REGION Network 7: 380A1 FB
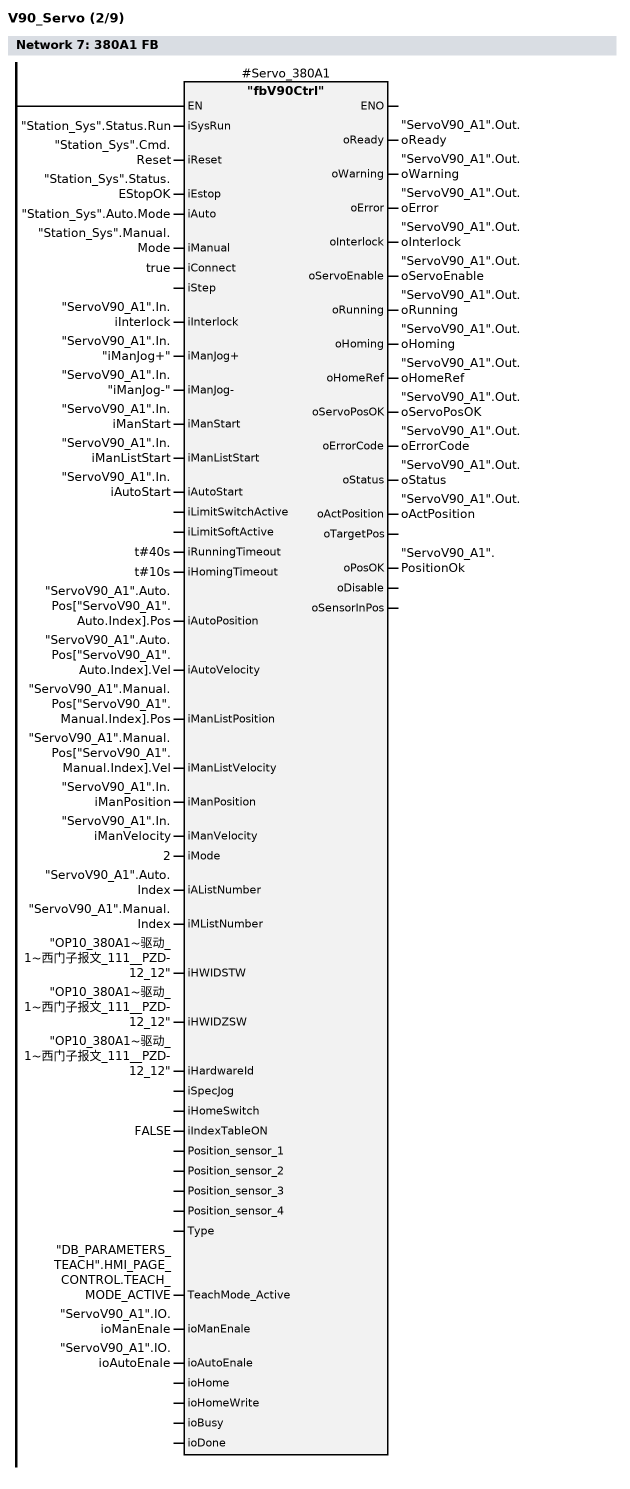
   RUNG wire#powerrail
      #Servo_380A1(iSysRun := "Station_Sys".Status.Run, iReset := "Station_Sys".Cmd.Reset, iEstop := "Station_Sys".Status.EStopOK, iAuto := "Station_Sys".Auto.Mode, iManual := "Station_Sys".Manual.Mode, iConnect := true, iStep :=, iInterlock := "ServoV90_A1".In.iInterlock, "iManJog+" := "ServoV90_A1".In."iManJog+", "iManJog-" := "ServoV90_A1".In."iManJog-", iManStart := "ServoV90_A1".In.iManStart, iManListStart := "ServoV90_A1".In.iManListStart, iAutoStart := "ServoV90_A1".In.iAutoStart, iLimitSwitchActive :=, iLimitSoftActive :=, iRunningTimeout := t#40s, iHomingTimeout := t#10s, iAutoPosition := "ServoV90_A1".Auto.Pos["ServoV90_A1".Auto.Index].Pos, iAutoVelocity := "ServoV90_A1".Auto.Pos["ServoV90_A1".Auto.Index].Vel, iManListPosition := "ServoV90_A1".Manual.Pos["ServoV90_A1".Manual.Index].Pos, iManListVelocity := "ServoV90_A1".Manual.Pos["ServoV90_A1".Manual.Index].Vel, iManPosition := "ServoV90_A1".In.iManPosition, iManVelocity := "ServoV90_A1".In.iManVelocity, iMode := 2, iAListNumber := "ServoV90_A1".Auto.Index, iMListNumber := "ServoV90_A1".Manual.Index, iHWIDSTW := "OP10_380A1~驱动_1~西门子报文_111__PZD-12_12", iHWIDZSW := "OP10_380A1~驱动_1~西门子报文_111__PZD-12_12", iHardwareId := "OP10_380A1~驱动_1~西门子报文_111__PZD-12_12", iSpecJog :=, iHomeSwitch :=, iIndexTableON := FALSE, Position_sensor_1 :=, Position_sensor_2 :=, Position_sensor_3 :=, Position_sensor_4 :=, "Type" :=, TeachMode_Active := "DB_PARAMETERS_TEACH".HMI_PAGE_CONTROL.TEACH_MODE_ACTIVE, ioManEnale := "ServoV90_A1".IO.ioManEnale, ioAutoEnale := "ServoV90_A1".IO.ioAutoEnale, ioHome :=, ioHomeWrite :=, ioBusy :=, ioDone :=, oReady => "ServoV90_A1".Out.oReady, oWarning => "ServoV90_A1".Out.oWarning, oError => "ServoV90_A1".Out.oError, oInterlock => "ServoV90_A1".Out.oInterlock, oServoEnable => "ServoV90_A1".Out.oServoEnable, oRunning => "ServoV90_A1".Out.oRunning, oHoming => "ServoV90_A1".Out.oHoming, oHomeRef => "ServoV90_A1".Out.oHomeRef, oServoPosOK => "ServoV90_A1".Out.oServoPosOK, oErrorCode => "ServoV90_A1".Out.oErrorCode, oStatus => "ServoV90_A1".Out.oStatus, oActPosition => "ServoV90_A1".Out.oActPosition, oTargetPos =>, oPosOK => "ServoV90_A1".PositionOk, oDisable =>, oSensorInPos =>)
   END_RUNG
   // the same network as SCL:
   #Servo_380A1(iSysRun := "Station_Sys".Status.Run,   // "fbV90Ctrl"
                iReset := "Station_Sys".Cmd.Reset,
                iEstop := "Station_Sys".Status.EStopOK,
                iAuto := "Station_Sys".Auto.Mode,
                iManual := "Station_Sys".Manual.Mode,
                iConnect := true,
                iInterlock := "ServoV90_A1".In.iInterlock,
                "iManJog+" := "ServoV90_A1".In."iManJog+",
                "iManJog-" := "ServoV90_A1".In."iManJog-",
                iManStart := "ServoV90_A1".In.iManStart,
                iManListStart := "ServoV90_A1".In.iManListStart,
                iAutoStart := "ServoV90_A1".In.iAutoStart,
                iRunningTimeout := t#40s,
                iHomingTimeout := t#10s,
                iAutoPosition := "ServoV90_A1".Auto.Pos["ServoV90_A1".Auto.Index].Pos,
                iAutoVelocity := "ServoV90_A1".Auto.Pos["ServoV90_A1".Auto.Index].Vel,
                iManListPosition := "ServoV90_A1".Manual.Pos["ServoV90_A1".Manual.Index].Pos,
                iManListVelocity := "ServoV90_A1".Manual.Pos["ServoV90_A1".Manual.Index].Vel,
                iManPosition := "ServoV90_A1".In.iManPosition,
                iManVelocity := "ServoV90_A1".In.iManVelocity,
                iMode := 2,
                iAListNumber := "ServoV90_A1".Auto.Index,
                iMListNumber := "ServoV90_A1".Manual.Index,
                iHWIDSTW := "OP10_380A1~驱动_1~西门子报文_111__PZD-12_12",
                iHWIDZSW := "OP10_380A1~驱动_1~西门子报文_111__PZD-12_12",
                iHardwareId := "OP10_380A1~驱动_1~西门子报文_111__PZD-12_12",
                iIndexTableON := FALSE,
                TeachMode_Active := "DB_PARAMETERS_TEACH".HMI_PAGE_CONTROL.TEACH_MODE_ACTIVE,
                ioManEnale := "ServoV90_A1".IO.ioManEnale,
                ioAutoEnale := "ServoV90_A1".IO.ioAutoEnale,
                oReady => "ServoV90_A1".Out.oReady,
                oWarning => "ServoV90_A1".Out.oWarning,
                oError => "ServoV90_A1".Out.oError,
                oInterlock => "ServoV90_A1".Out.oInterlock,
                oServoEnable => "ServoV90_A1".Out.oServoEnable,
                oRunning => "ServoV90_A1".Out.oRunning,
                oHoming => "ServoV90_A1".Out.oHoming,
                oHomeRef => "ServoV90_A1".Out.oHomeRef,
                oServoPosOK => "ServoV90_A1".Out.oServoPosOK,
                oErrorCode => "ServoV90_A1".Out.oErrorCode,
                oStatus => "ServoV90_A1".Out.oStatus,
                oActPosition => "ServoV90_A1".Out.oActPosition,
                oPosOK => "ServoV90_A1".PositionOk);
END_REGION

REGION Network 8 (SCL): 故障显示 / Fault indication
   //"ST70_DeviceError".Servo1.ServoDriverError := "ServoV90_A1".Out.oError;
END_REGION

REGION Network 9: <<<<<<<<<<<<<<<<<<<<<381A1 Servo>>>>>>>>>>>>>>>>>>>>>>>>>
END_REGION

REGION Network 10: negtive motion/action/...automaticly
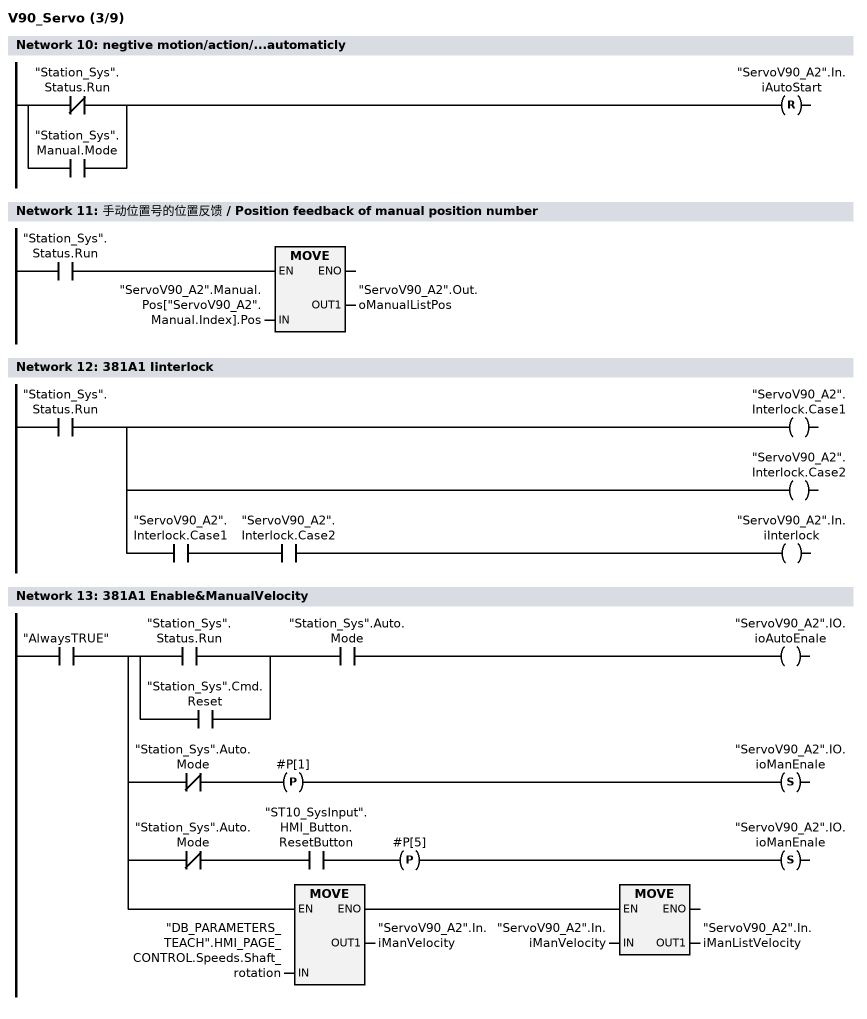
   RUNG wire#powerrail
      I_Contact( "Station_Sys".Status.Run )
      wire#w1
      R_Coil( "ServoV90_A2".In.iAutoStart )
   END_RUNG
   RUNG wire#powerrail
      Contact( "Station_Sys".Manual.Mode )
   END_RUNG wire#w1
   // the same network as SCL:
   IF NOT "Station_Sys".Status.Run OR "Station_Sys".Manual.Mode THEN
       "ServoV90_A2".In.iAutoStart := FALSE;
   END_IF;
END_REGION

REGION Network 11: 手动位置号的位置反馈 / Position feedback of manual position number
   RUNG wire#powerrail
      Contact( "Station_Sys".Status.Run )
      Move(in := "ServoV90_A2".Manual.Pos["ServoV90_A2".Manual.Index].Pos, out1 => "ServoV90_A2".Out.oManualListPos)
   END_RUNG
   // the same network as SCL:
   IF "Station_Sys".Status.Run THEN
       "ServoV90_A2".Out.oManualListPos := "ServoV90_A2".Manual.Pos["ServoV90_A2".Manual.Index].Pos;
   END_IF;
END_REGION

REGION Network 12: 381A1 Iinterlock
   RUNG wire#powerrail
      Contact( "Station_Sys".Status.Run )
      wire#w1
      Coil( "ServoV90_A2".Interlock.Case1 )
   END_RUNG
   RUNG wire#w1
      Coil( "ServoV90_A2".Interlock.Case2 )
   END_RUNG
   RUNG wire#w1
      Contact( "ServoV90_A2".Interlock.Case1 )
      Contact( "ServoV90_A2".Interlock.Case2 )
      Coil( "ServoV90_A2".In.iInterlock )
   END_RUNG
   // the same network as SCL:
   "ServoV90_A2".Interlock.Case1 := "Station_Sys".Status.Run;
   "ServoV90_A2".Interlock.Case2 := "Station_Sys".Status.Run;
   "ServoV90_A2".In.iInterlock := "Station_Sys".Status.Run AND "ServoV90_A2".Interlock.Case1 AND "ServoV90_A2".Interlock.Case2;
END_REGION

REGION Network 13: 381A1 Enable&ManualVelocity
   RUNG wire#powerrail
      Contact( "AlwaysTRUE" )
      wire#w1
      Contact( "Station_Sys".Status.Run )
      wire#w2
      Contact( "Station_Sys".Auto.Mode )
      Coil( "ServoV90_A2".IO.ioAutoEnale )
   END_RUNG
   RUNG wire#w1
      Contact( "Station_Sys".Cmd.Reset )
   END_RUNG wire#w2
   RUNG wire#w1
      I_Contact( "Station_Sys".Auto.Mode )
      P_Trig( #P[1] )
      S_Coil( "ServoV90_A2".IO.ioManEnale )
   END_RUNG
   RUNG wire#w1
      I_Contact( "Station_Sys".Auto.Mode )
      Contact( "ST10_SysInput".HMI_Button.ResetButton )
      P_Trig( #P[5] )
      S_Coil( "ServoV90_A2".IO.ioManEnale )
   END_RUNG
   RUNG wire#w1
      Move(in := "DB_PARAMETERS_TEACH".HMI_PAGE_CONTROL.Speeds.Shaft_rotation, out1 => "ServoV90_A2".In.iManVelocity)
      Move(in := "ServoV90_A2".In.iManVelocity, out1 => "ServoV90_A2".In.iManListVelocity)
   END_RUNG
   // the same network as SCL:
   "ServoV90_A2".IO.ioAutoEnale := "AlwaysTRUE" AND ("Station_Sys".Status.Run OR "Station_Sys".Cmd.Reset) AND "Station_Sys".Auto.Mode;
   #_w1 := "AlwaysTRUE" AND NOT "Station_Sys".Auto.Mode;
   #_w2 := #_w1 AND NOT #P[1];   // rising edge
   #P[1] := #_w1;
   IF #_w2 THEN "ServoV90_A2".IO.ioManEnale := TRUE; END_IF;
   #_w3 := "AlwaysTRUE" AND NOT "Station_Sys".Auto.Mode AND "ST10_SysInput".HMI_Button.ResetButton;
   #_w4 := #_w3 AND NOT #P[5];   // rising edge
   #P[5] := #_w3;
   IF #_w4 THEN "ServoV90_A2".IO.ioManEnale := TRUE; END_IF;
   IF "AlwaysTRUE" THEN
       "ServoV90_A2".In.iManVelocity := "DB_PARAMETERS_TEACH".HMI_PAGE_CONTROL.Speeds.Shaft_rotation;
       "ServoV90_A2".In.iManListVelocity := "ServoV90_A2".In.iManVelocity;
   END_IF;
END_REGION

REGION Network 14 (SCL): 381A1 RecipePosition
    IF "Station_Sys".Status.Run THEN
        "ServoV90_A2".Manual.Pos[1].Pos := "ServoV90_A2".Auto.Pos[1].Pos := REAL_TO_DINT("Parameter".AxisRun.Axis[2].Pos1.Position*1000);
       "ServoV90_A2".Manual.Pos[1].Vel := "ServoV90_A2".Auto.Pos[1].Vel := "Parameter".AxisRun.Axis[2].Pos1.Speed;

       "ServoV90_A2".Manual.Pos[2].Pos := "ServoV90_A2".Auto.Pos[2].Pos := REAL_TO_DINT("Parameter".AxisRun.Axis[2].Pos2.Position*1000);
       "ServoV90_A2".Manual.Pos[2].Vel := "ServoV90_A2".Auto.Pos[2].Vel := "Parameter".AxisRun.Axis[2].Pos2.Speed;

       "ServoV90_A2".Manual.Pos[3].Pos := "ServoV90_A2".Auto.Pos[3].Pos := REAL_TO_DINT("Parameter".AxisRun.Axis[2].Pos3.Position*1000);
       "ServoV90_A2".Manual.Pos[3].Vel := "ServoV90_A2".Auto.Pos[3].Vel := "Parameter".AxisRun.Axis[2].Pos3.Speed;

       "ServoV90_A2".Manual.Pos[4].Pos := "ServoV90_A2".Auto.Pos[4].Pos := REAL_TO_DINT("Parameter".AxisRun.Axis[2].Pos4.Position*1000);
       "ServoV90_A2".Manual.Pos[4].Vel := "ServoV90_A2".Auto.Pos[4].Vel := "Parameter".AxisRun.Axis[2].Pos4.Speed;

       "ServoV90_A2".Manual.Pos[5].Pos := "ServoV90_A2".Auto.Pos[5].Pos := REAL_TO_DINT("Parameter".AxisRun.Axis[2].Pos5.Position*1000);
       "ServoV90_A2".Manual.Pos[5].Vel := "ServoV90_A2".Auto.Pos[5].Vel := "Parameter".AxisRun.Axis[2].Pos5.Speed;

       "ServoV90_A2".Manual.Pos[6].Pos := "ServoV90_A2".Auto.Pos[6].Pos := REAL_TO_DINT("Parameter".AxisRun.Axis[2].Pos6.Position*1000);
       "ServoV90_A2".Manual.Pos[6].Vel := "ServoV90_A2".Auto.Pos[6].Vel := "Parameter".AxisRun.Axis[2].Pos6.Speed;

       "ServoV90_A2".Manual.Pos[7].Pos := "ServoV90_A2".Auto.Pos[7].Pos := REAL_TO_DINT("Parameter".AxisRun.Axis[2].Pos7.Position*1000);
       "ServoV90_A2".Manual.Pos[7].Vel := "ServoV90_A2".Auto.Pos[7].Vel := "Parameter".AxisRun.Axis[2].Pos7.Speed;

       "ServoV90_A2".Manual.Pos[8].Pos := "ServoV90_A2".Auto.Pos[8].Pos := REAL_TO_DINT("Parameter".AxisRun.Axis[2].Pos8.Position*1000);
       "ServoV90_A2".Manual.Pos[8].Vel := "ServoV90_A2".Auto.Pos[8].Vel := "Parameter".AxisRun.Axis[2].Pos8.Speed;

       "ServoV90_A2".Manual.Pos[9].Pos := "ServoV90_A2".Auto.Pos[9].Pos := REAL_TO_DINT("Parameter".AxisRun.Axis[2].Pos9.Position*1000);
       "ServoV90_A2".Manual.Pos[9].Vel := "ServoV90_A2".Auto.Pos[9].Vel := "Parameter".AxisRun.Axis[2].Pos9.Speed;

       "ServoV90_A2".Manual.Pos[10].Pos := "ServoV90_A2".Auto.Pos[10].Pos := REAL_TO_DINT("Parameter".AxisRun.Axis[2].Pos10.Position*1000);
       "ServoV90_A2".Manual.Pos[10].Vel := "ServoV90_A2".Auto.Pos[10].Vel := "Parameter".AxisRun.Axis[2].Pos10.Speed;
   END_IF;
END_REGION

REGION Network 15: 381A1 FB
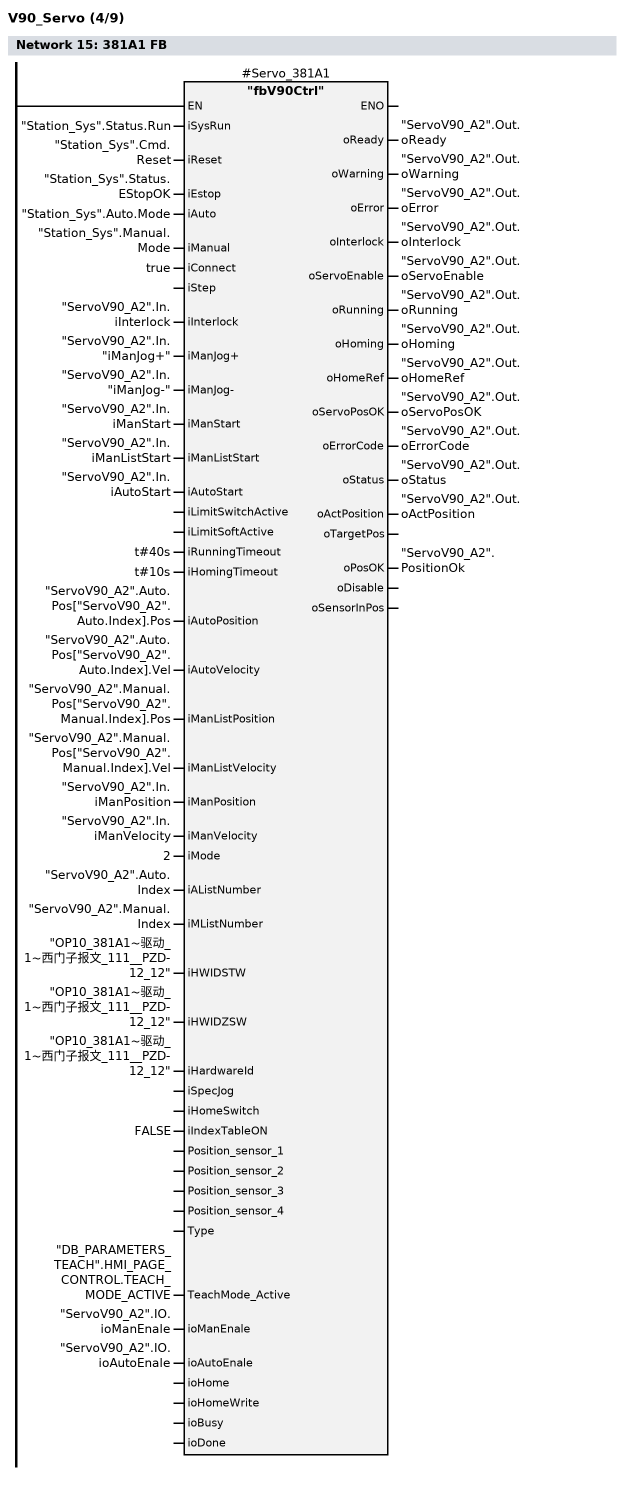
   RUNG wire#powerrail
      #Servo_381A1(iSysRun := "Station_Sys".Status.Run, iReset := "Station_Sys".Cmd.Reset, iEstop := "Station_Sys".Status.EStopOK, iAuto := "Station_Sys".Auto.Mode, iManual := "Station_Sys".Manual.Mode, iConnect := true, iStep :=, iInterlock := "ServoV90_A2".In.iInterlock, "iManJog+" := "ServoV90_A2".In."iManJog+", "iManJog-" := "ServoV90_A2".In."iManJog-", iManStart := "ServoV90_A2".In.iManStart, iManListStart := "ServoV90_A2".In.iManListStart, iAutoStart := "ServoV90_A2".In.iAutoStart, iLimitSwitchActive :=, iLimitSoftActive :=, iRunningTimeout := t#40s, iHomingTimeout := t#10s, iAutoPosition := "ServoV90_A2".Auto.Pos["ServoV90_A2".Auto.Index].Pos, iAutoVelocity := "ServoV90_A2".Auto.Pos["ServoV90_A2".Auto.Index].Vel, iManListPosition := "ServoV90_A2".Manual.Pos["ServoV90_A2".Manual.Index].Pos, iManListVelocity := "ServoV90_A2".Manual.Pos["ServoV90_A2".Manual.Index].Vel, iManPosition := "ServoV90_A2".In.iManPosition, iManVelocity := "ServoV90_A2".In.iManVelocity, iMode := 2, iAListNumber := "ServoV90_A2".Auto.Index, iMListNumber := "ServoV90_A2".Manual.Index, iHWIDSTW := "OP10_381A1~驱动_1~西门子报文_111__PZD-12_12", iHWIDZSW := "OP10_381A1~驱动_1~西门子报文_111__PZD-12_12", iHardwareId := "OP10_381A1~驱动_1~西门子报文_111__PZD-12_12", iSpecJog :=, iHomeSwitch :=, iIndexTableON := FALSE, Position_sensor_1 :=, Position_sensor_2 :=, Position_sensor_3 :=, Position_sensor_4 :=, "Type" :=, TeachMode_Active := "DB_PARAMETERS_TEACH".HMI_PAGE_CONTROL.TEACH_MODE_ACTIVE, ioManEnale := "ServoV90_A2".IO.ioManEnale, ioAutoEnale := "ServoV90_A2".IO.ioAutoEnale, ioHome :=, ioHomeWrite :=, ioBusy :=, ioDone :=, oReady => "ServoV90_A2".Out.oReady, oWarning => "ServoV90_A2".Out.oWarning, oError => "ServoV90_A2".Out.oError, oInterlock => "ServoV90_A2".Out.oInterlock, oServoEnable => "ServoV90_A2".Out.oServoEnable, oRunning => "ServoV90_A2".Out.oRunning, oHoming => "ServoV90_A2".Out.oHoming, oHomeRef => "ServoV90_A2".Out.oHomeRef, oServoPosOK => "ServoV90_A2".Out.oServoPosOK, oErrorCode => "ServoV90_A2".Out.oErrorCode, oStatus => "ServoV90_A2".Out.oStatus, oActPosition => "ServoV90_A2".Out.oActPosition, oTargetPos =>, oPosOK => "ServoV90_A2".PositionOk, oDisable =>, oSensorInPos =>)
   END_RUNG
   // the same network as SCL:
   #Servo_381A1(iSysRun := "Station_Sys".Status.Run,   // "fbV90Ctrl"
                iReset := "Station_Sys".Cmd.Reset,
                iEstop := "Station_Sys".Status.EStopOK,
                iAuto := "Station_Sys".Auto.Mode,
                iManual := "Station_Sys".Manual.Mode,
                iConnect := true,
                iInterlock := "ServoV90_A2".In.iInterlock,
                "iManJog+" := "ServoV90_A2".In."iManJog+",
                "iManJog-" := "ServoV90_A2".In."iManJog-",
                iManStart := "ServoV90_A2".In.iManStart,
                iManListStart := "ServoV90_A2".In.iManListStart,
                iAutoStart := "ServoV90_A2".In.iAutoStart,
                iRunningTimeout := t#40s,
                iHomingTimeout := t#10s,
                iAutoPosition := "ServoV90_A2".Auto.Pos["ServoV90_A2".Auto.Index].Pos,
                iAutoVelocity := "ServoV90_A2".Auto.Pos["ServoV90_A2".Auto.Index].Vel,
                iManListPosition := "ServoV90_A2".Manual.Pos["ServoV90_A2".Manual.Index].Pos,
                iManListVelocity := "ServoV90_A2".Manual.Pos["ServoV90_A2".Manual.Index].Vel,
                iManPosition := "ServoV90_A2".In.iManPosition,
                iManVelocity := "ServoV90_A2".In.iManVelocity,
                iMode := 2,
                iAListNumber := "ServoV90_A2".Auto.Index,
                iMListNumber := "ServoV90_A2".Manual.Index,
                iHWIDSTW := "OP10_381A1~驱动_1~西门子报文_111__PZD-12_12",
                iHWIDZSW := "OP10_381A1~驱动_1~西门子报文_111__PZD-12_12",
                iHardwareId := "OP10_381A1~驱动_1~西门子报文_111__PZD-12_12",
                iIndexTableON := FALSE,
                TeachMode_Active := "DB_PARAMETERS_TEACH".HMI_PAGE_CONTROL.TEACH_MODE_ACTIVE,
                ioManEnale := "ServoV90_A2".IO.ioManEnale,
                ioAutoEnale := "ServoV90_A2".IO.ioAutoEnale,
                oReady => "ServoV90_A2".Out.oReady,
                oWarning => "ServoV90_A2".Out.oWarning,
                oError => "ServoV90_A2".Out.oError,
                oInterlock => "ServoV90_A2".Out.oInterlock,
                oServoEnable => "ServoV90_A2".Out.oServoEnable,
                oRunning => "ServoV90_A2".Out.oRunning,
                oHoming => "ServoV90_A2".Out.oHoming,
                oHomeRef => "ServoV90_A2".Out.oHomeRef,
                oServoPosOK => "ServoV90_A2".Out.oServoPosOK,
                oErrorCode => "ServoV90_A2".Out.oErrorCode,
                oStatus => "ServoV90_A2".Out.oStatus,
                oActPosition => "ServoV90_A2".Out.oActPosition,
                oPosOK => "ServoV90_A2".PositionOk);
END_REGION

REGION Network 16 (SCL): 故障显示 / Fault indication
   //"ST70_DeviceError".Servo2.ServoDriverError := "ServoV90_A2".Out.oError;
   //

   "ServoV90_A3".Auto.Index := "ServoV90_A3".Auto.Index;
END_REGION

REGION Network 17: <<<<<<<<<<<<<<<<<<<<<382A1 Servo>>>>>>>>>>>>>>>>>>>>>>>>>
END_REGION

REGION Network 18: <<<<<<<<<<<<<<<<<<<<<382A1 Servo>>>>>>>>>>>>>>>>>>>>>>>>> / $$$$####### NEW TECHNOLOGY OBJECTS #################
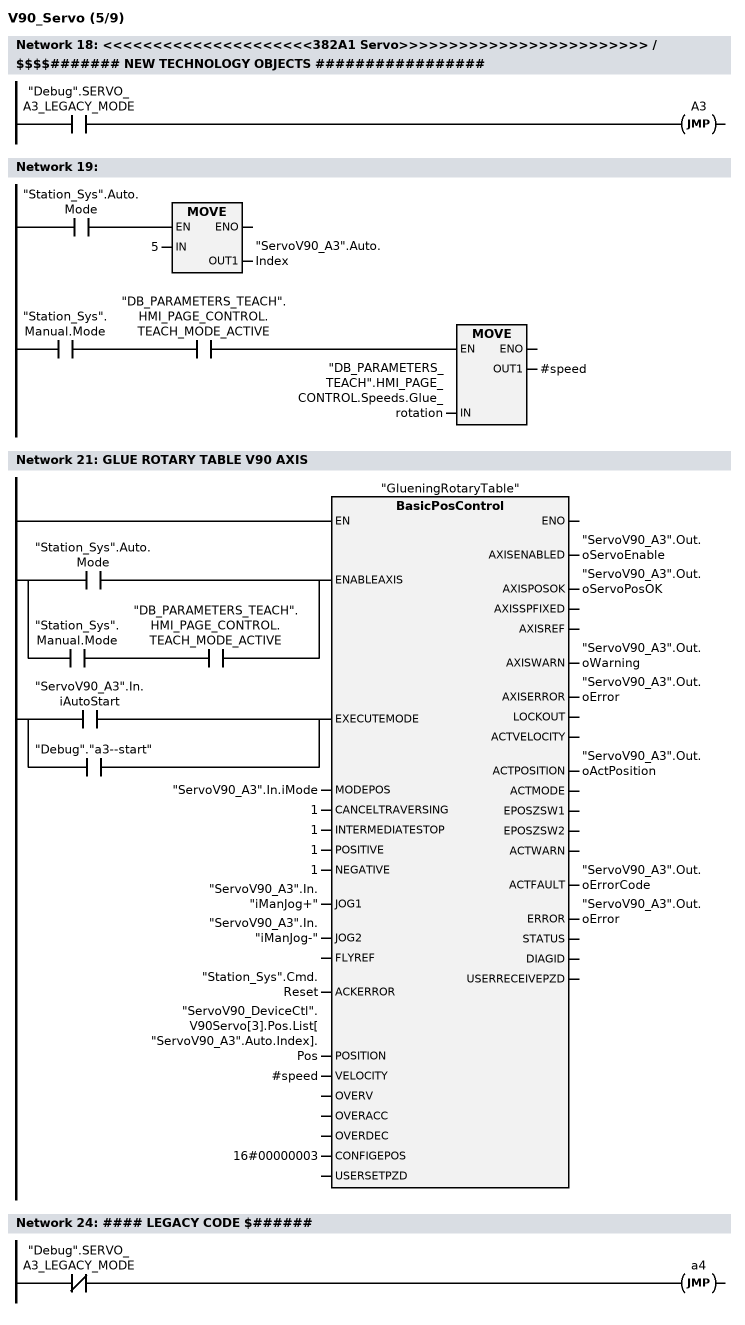
   RUNG wire#powerrail
      Contact( "Debug".SERVO_A3_LEGACY_MODE )
      JumpCoil( A3 )
   END_RUNG
   // the same network as SCL:
   IF "Debug".SERVO_A3_LEGACY_MODE THEN GOTO A3; END_IF;
END_REGION

REGION Network 19
   RUNG wire#powerrail
      Contact( "Station_Sys".Auto.Mode )
      Move(in := 5, out1 => "ServoV90_A3".Auto.Index)
   END_RUNG
   RUNG wire#powerrail
      Contact( "Station_Sys".Manual.Mode )
      Contact( "DB_PARAMETERS_TEACH".HMI_PAGE_CONTROL.TEACH_MODE_ACTIVE )
      Move(in := "DB_PARAMETERS_TEACH".HMI_PAGE_CONTROL.Speeds.Glue_rotation, out1 => #speed)
   END_RUNG
   // the same network as SCL:
   IF "Station_Sys".Auto.Mode THEN "ServoV90_A3".Auto.Index := 5; END_IF;
   IF "Station_Sys".Manual.Mode AND "DB_PARAMETERS_TEACH".HMI_PAGE_CONTROL.TEACH_MODE_ACTIVE THEN
       #speed := "DB_PARAMETERS_TEACH".HMI_PAGE_CONTROL.Speeds.Glue_rotation;
   END_IF;
END_REGION

REGION Network 21: GLUE ROTARY TABLE V90 AXIS
   RUNG wire#powerrail
      "GlueningRotaryTable".BasicPosControl(EnableAxis := wire#w1, ExecuteMode := wire#w2, ModePos := "ServoV90_A3".In.iMode, CancelTraversing := 1, IntermediateStop := 1, Positive := 1, Negative := 1, Jog1 := "ServoV90_A3".In."iManJog+", Jog2 := "ServoV90_A3".In."iManJog-", FlyRef :=, AckError := "Station_Sys".Cmd.Reset, Position := "ServoV90_DeviceCtl".V90Servo[3].Pos.List["ServoV90_A3".Auto.Index].Pos, Velocity := #speed, OverV :=, OverAcc :=, OverDec :=, ConfigEPos := 16#00000003, UserSetPZD :=, AxisEnabled => "ServoV90_A3".Out.oServoEnable, AxisPosOk => "ServoV90_A3".Out.oServoPosOK, AxisSpFixed =>, AxisRef =>, AxisWarn => "ServoV90_A3".Out.oWarning, AxisError => "ServoV90_A3".Out.oError, Lockout =>, ActVelocity =>, ActPosition => "ServoV90_A3".Out.oActPosition, ActMode =>, EPosZSW1 =>, EPosZSW2 =>, ActWarn =>, ActFault => "ServoV90_A3".Out.oErrorCode, Error => "ServoV90_A3".Out.oError, Status =>, DiagId =>, UserReceivePZD =>)
   END_RUNG
   RUNG wire#powerrail
      Contact( "Station_Sys".Auto.Mode )
   END_RUNG wire#w1
   RUNG wire#powerrail
      Contact( "Station_Sys".Manual.Mode )
      Contact( "DB_PARAMETERS_TEACH".HMI_PAGE_CONTROL.TEACH_MODE_ACTIVE )
   END_RUNG wire#w1
   RUNG wire#powerrail
      Contact( "ServoV90_A3".In.iAutoStart )
   END_RUNG wire#w2
   RUNG wire#powerrail
      Contact( "Debug"."a3--start" )
   END_RUNG wire#w2
   // the same network as SCL:
   "GlueningRotaryTable"(EnableAxis := "Station_Sys".Auto.Mode OR ("Station_Sys".Manual.Mode AND "DB_PARAMETERS_TEACH".HMI_PAGE_CONTROL.TEACH_MODE_ACTIVE),   // BasicPosControl
                         ExecuteMode := "ServoV90_A3".In.iAutoStart OR "Debug"."a3--start",
                         ModePos := "ServoV90_A3".In.iMode,
                         CancelTraversing := 1,
                         IntermediateStop := 1,
                         Positive := 1,
                         Negative := 1,
                         Jog1 := "ServoV90_A3".In."iManJog+",
                         Jog2 := "ServoV90_A3".In."iManJog-",
                         AckError := "Station_Sys".Cmd.Reset,
                         Position := "ServoV90_DeviceCtl".V90Servo[3].Pos.List["ServoV90_A3".Auto.Index].Pos,
                         Velocity := #speed,
                         ConfigEPos := 16#00000003,
                         AxisEnabled => "ServoV90_A3".Out.oServoEnable,
                         AxisPosOk => "ServoV90_A3".Out.oServoPosOK,
                         AxisWarn => "ServoV90_A3".Out.oWarning,
                         AxisError => "ServoV90_A3".Out.oError,
                         ActPosition => "ServoV90_A3".Out.oActPosition,
                         ActFault => "ServoV90_A3".Out.oErrorCode,
                         Error => "ServoV90_A3".Out.oError);
END_REGION

REGION Network 23: <<<<<<<<<<<<<<<<<<<<<382A1 Servo>>>>>>>>>>>>>>>>>>>>>>>>> / ################# ##################################
END_REGION

REGION Network 24: #### LEGACY CODE $######
   RUNG wire#powerrail
      I_Contact( "Debug".SERVO_A3_LEGACY_MODE )
      JumpCoil( a4 )
   END_RUNG
   // the same network as SCL:
   IF NOT "Debug".SERVO_A3_LEGACY_MODE THEN GOTO a4; END_IF;
END_REGION

REGION Network 25: negtive motion/action/...automaticly
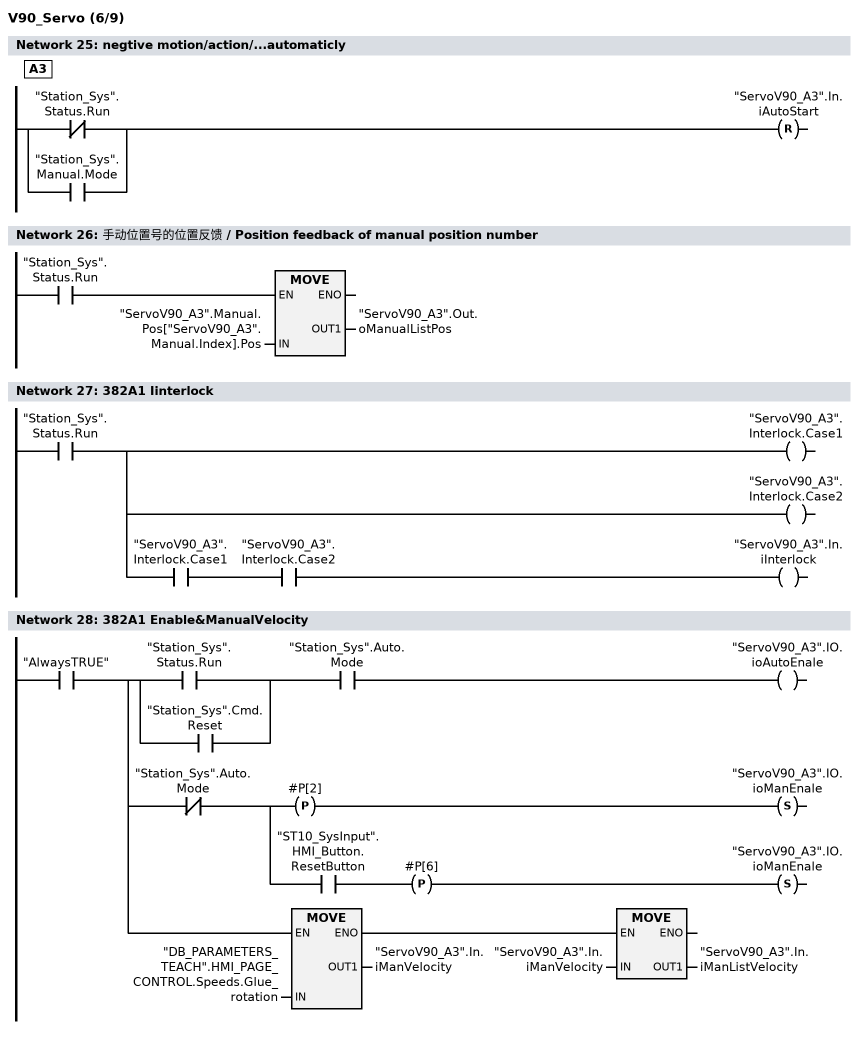
   Label( A3 )
   RUNG wire#powerrail
      I_Contact( "Station_Sys".Status.Run )
      wire#w1
      R_Coil( "ServoV90_A3".In.iAutoStart )
   END_RUNG
   RUNG wire#powerrail
      Contact( "Station_Sys".Manual.Mode )
   END_RUNG wire#w1
   // the same network as SCL:
   A3:
   IF NOT "Station_Sys".Status.Run OR "Station_Sys".Manual.Mode THEN
       "ServoV90_A3".In.iAutoStart := FALSE;
   END_IF;
END_REGION

REGION Network 26: 手动位置号的位置反馈 / Position feedback of manual position number
   RUNG wire#powerrail
      Contact( "Station_Sys".Status.Run )
      Move(in := "ServoV90_A3".Manual.Pos["ServoV90_A3".Manual.Index].Pos, out1 => "ServoV90_A3".Out.oManualListPos)
   END_RUNG
   // the same network as SCL:
   IF "Station_Sys".Status.Run THEN
       "ServoV90_A3".Out.oManualListPos := "ServoV90_A3".Manual.Pos["ServoV90_A3".Manual.Index].Pos;
   END_IF;
END_REGION

REGION Network 27: 382A1 Iinterlock
   RUNG wire#powerrail
      Contact( "Station_Sys".Status.Run )
      wire#w1
      Coil( "ServoV90_A3".Interlock.Case1 )
   END_RUNG
   RUNG wire#w1
      Coil( "ServoV90_A3".Interlock.Case2 )
   END_RUNG
   RUNG wire#w1
      Contact( "ServoV90_A3".Interlock.Case1 )
      Contact( "ServoV90_A3".Interlock.Case2 )
      Coil( "ServoV90_A3".In.iInterlock )
   END_RUNG
   // the same network as SCL:
   "ServoV90_A3".Interlock.Case1 := "Station_Sys".Status.Run;
   "ServoV90_A3".Interlock.Case2 := "Station_Sys".Status.Run;
   "ServoV90_A3".In.iInterlock := "Station_Sys".Status.Run AND "ServoV90_A3".Interlock.Case1 AND "ServoV90_A3".Interlock.Case2;
END_REGION

REGION Network 28: 382A1 Enable&ManualVelocity
   RUNG wire#powerrail
      Contact( "AlwaysTRUE" )
      wire#w1
      Contact( "Station_Sys".Status.Run )
      wire#w2
      Contact( "Station_Sys".Auto.Mode )
      Coil( "ServoV90_A3".IO.ioAutoEnale )
   END_RUNG
   RUNG wire#w1
      Contact( "Station_Sys".Cmd.Reset )
   END_RUNG wire#w2
   RUNG wire#w1
      I_Contact( "Station_Sys".Auto.Mode )
      wire#w3
      P_Trig( #P[2] )
      S_Coil( "ServoV90_A3".IO.ioManEnale )
   END_RUNG
   RUNG wire#w3
      Contact( "ST10_SysInput".HMI_Button.ResetButton )
      P_Trig( #P[6] )
      S_Coil( "ServoV90_A3".IO.ioManEnale )
   END_RUNG
   RUNG wire#w1
      Move(in := "DB_PARAMETERS_TEACH".HMI_PAGE_CONTROL.Speeds.Glue_rotation, out1 => "ServoV90_A3".In.iManVelocity)
      Move(in := "ServoV90_A3".In.iManVelocity, out1 => "ServoV90_A3".In.iManListVelocity)
   END_RUNG
   // the same network as SCL:
   "ServoV90_A3".IO.ioAutoEnale := "AlwaysTRUE" AND ("Station_Sys".Status.Run OR "Station_Sys".Cmd.Reset) AND "Station_Sys".Auto.Mode;
   #_w1 := "AlwaysTRUE" AND NOT "Station_Sys".Auto.Mode;
   #_w2 := #_w1 AND NOT #P[2];   // rising edge
   #P[2] := #_w1;
   IF #_w2 THEN "ServoV90_A3".IO.ioManEnale := TRUE; END_IF;
   #_w3 := #_w1 AND "ST10_SysInput".HMI_Button.ResetButton;
   #_w4 := #_w3 AND NOT #P[6];   // rising edge
   #P[6] := #_w3;
   IF #_w4 THEN "ServoV90_A3".IO.ioManEnale := TRUE; END_IF;
   IF "AlwaysTRUE" THEN
       "ServoV90_A3".In.iManVelocity := "DB_PARAMETERS_TEACH".HMI_PAGE_CONTROL.Speeds.Glue_rotation;
       "ServoV90_A3".In.iManListVelocity := "ServoV90_A3".In.iManVelocity;
   END_IF;
END_REGION

REGION Network 29 (SCL): 382A1 RecipePosition
    IF "Station_Sys".Status.Run THEN
        "ServoV90_A3".Manual.Pos[1].Pos := "ServoV90_A3".Auto.Pos[1].Pos := REAL_TO_DINT("Parameter".AxisRun.Axis[3].Pos1.Position*1000);
        "ServoV90_A3".Manual.Pos[1].Vel := "ServoV90_A3".Auto.Pos[1].Vel := "Parameter".AxisRun.Axis[3].Pos1.Speed;

        "ServoV90_A3".Manual.Pos[2].Pos := "ServoV90_A3".Auto.Pos[2].Pos := REAL_TO_DINT("Parameter".AxisRun.Axis[3].Pos2.Position*1000);
        "ServoV90_A3".Manual.Pos[2].Vel := "ServoV90_A3".Auto.Pos[2].Vel := "Parameter".AxisRun.Axis[3].Pos2.Speed;

        "ServoV90_A3".Manual.Pos[3].Pos := "ServoV90_A3".Auto.Pos[3].Pos := REAL_TO_DINT("Parameter".AxisRun.Axis[3].Pos3.Position*1000);
        "ServoV90_A3".Manual.Pos[3].Vel := "ServoV90_A3".Auto.Pos[3].Vel := "Parameter".AxisRun.Axis[3].Pos3.Speed;

        "ServoV90_A3".Manual.Pos[4].Pos := "ServoV90_A3".Auto.Pos[4].Pos := REAL_TO_DINT("Parameter".AxisRun.Axis[3].Pos4.Position*1000);
        "ServoV90_A3".Manual.Pos[4].Vel := "ServoV90_A3".Auto.Pos[4].Vel := "Parameter".AxisRun.Axis[3].Pos4.Speed;

        "ServoV90_A3".Manual.Pos[5].Pos := "ServoV90_A3".Auto.Pos[5].Pos := REAL_TO_DINT("Parameter".AxisRun.Axis[3].Pos5.Position*1000);
        "ServoV90_A3".Manual.Pos[5].Vel := "ServoV90_A3".Auto.Pos[5].Vel := "Parameter".AxisRun.Axis[3].Pos5.Speed;

        "ServoV90_A3".Manual.Pos[6].Pos := "ServoV90_A3".Auto.Pos[6].Pos := REAL_TO_DINT("Parameter".AxisRun.Axis[3].Pos6.Position*1000);
        "ServoV90_A3".Manual.Pos[6].Vel := "ServoV90_A3".Auto.Pos[6].Vel := "Parameter".AxisRun.Axis[3].Pos6.Speed;

        "ServoV90_A3".Manual.Pos[7].Pos := "ServoV90_A3".Auto.Pos[7].Pos := REAL_TO_DINT("Parameter".AxisRun.Axis[3].Pos7.Position*1000);
        "ServoV90_A3".Manual.Pos[7].Vel := "ServoV90_A3".Auto.Pos[7].Vel := "Parameter".AxisRun.Axis[3].Pos7.Speed;

        "ServoV90_A3".Manual.Pos[8].Pos := "ServoV90_A3".Auto.Pos[8].Pos := REAL_TO_DINT("Parameter".AxisRun.Axis[3].Pos8.Position*1000);
        "ServoV90_A3".Manual.Pos[8].Vel := "ServoV90_A3".Auto.Pos[8].Vel := "Parameter".AxisRun.Axis[3].Pos8.Speed;

        "ServoV90_A3".Manual.Pos[9].Pos := "ServoV90_A3".Auto.Pos[9].Pos := REAL_TO_DINT("Parameter".AxisRun.Axis[3].Pos9.Position*1000);
        "ServoV90_A3".Manual.Pos[9].Vel := "ServoV90_A3".Auto.Pos[9].Vel := "Parameter".AxisRun.Axis[3].Pos9.Speed;

        "ServoV90_A3".Manual.Pos[10].Pos := "ServoV90_A3".Auto.Pos[10].Pos := REAL_TO_DINT("Parameter".AxisRun.Axis[3].Pos10.Position*1000);
        "ServoV90_A3".Manual.Pos[10].Vel := "ServoV90_A3".Auto.Pos[10].Vel := "Parameter".AxisRun.Axis[3].Pos10.Speed;
   END_IF;
END_REGION

REGION Network 30: 382A1 FB
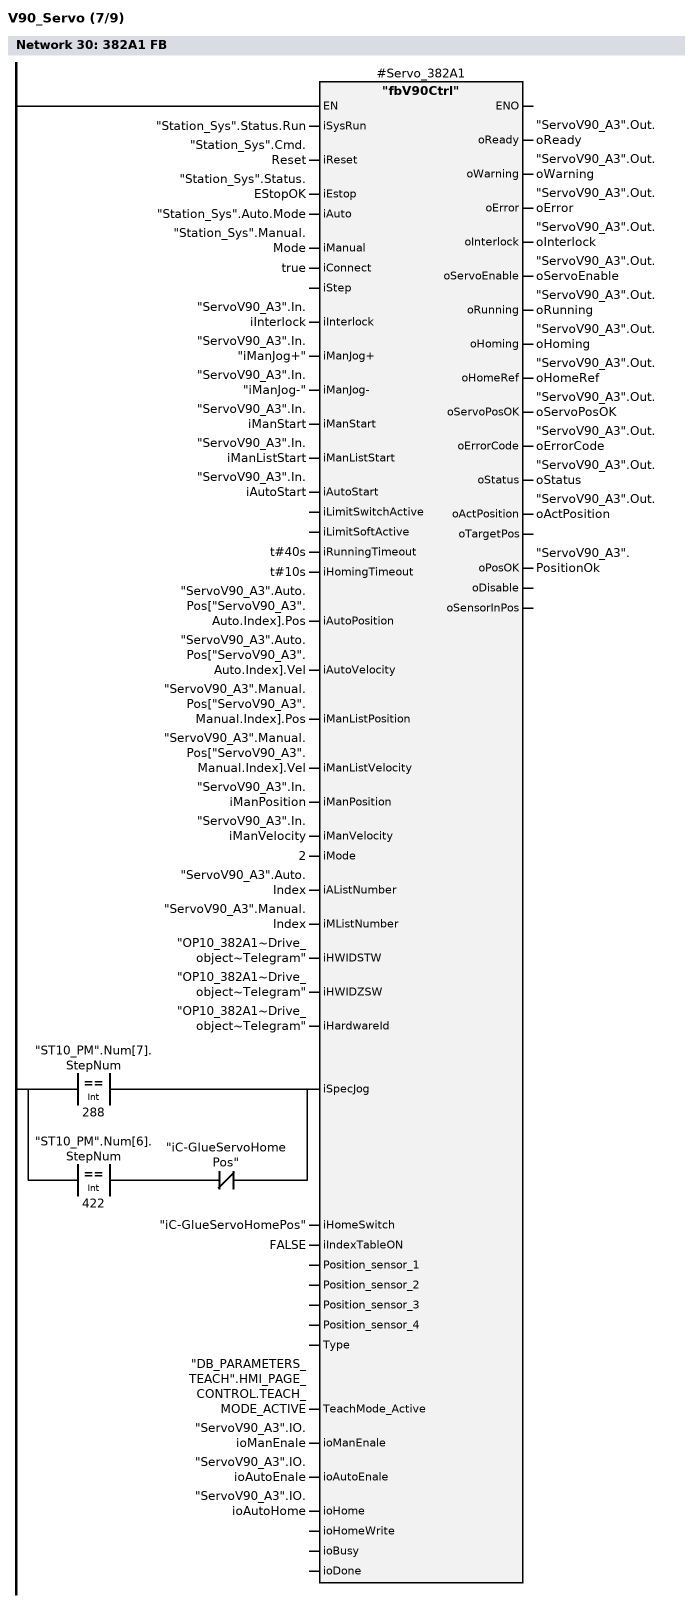
   RUNG wire#powerrail
      #Servo_382A1(iSpecJog := wire#w1, iSysRun := "Station_Sys".Status.Run, iReset := "Station_Sys".Cmd.Reset, iEstop := "Station_Sys".Status.EStopOK, iAuto := "Station_Sys".Auto.Mode, iManual := "Station_Sys".Manual.Mode, iConnect := true, iStep :=, iInterlock := "ServoV90_A3".In.iInterlock, "iManJog+" := "ServoV90_A3".In."iManJog+", "iManJog-" := "ServoV90_A3".In."iManJog-", iManStart := "ServoV90_A3".In.iManStart, iManListStart := "ServoV90_A3".In.iManListStart, iAutoStart := "ServoV90_A3".In.iAutoStart, iLimitSwitchActive :=, iLimitSoftActive :=, iRunningTimeout := t#40s, iHomingTimeout := t#10s, iAutoPosition := "ServoV90_A3".Auto.Pos["ServoV90_A3".Auto.Index].Pos, iAutoVelocity := "ServoV90_A3".Auto.Pos["ServoV90_A3".Auto.Index].Vel, iManListPosition := "ServoV90_A3".Manual.Pos["ServoV90_A3".Manual.Index].Pos, iManListVelocity := "ServoV90_A3".Manual.Pos["ServoV90_A3".Manual.Index].Vel, iManPosition := "ServoV90_A3".In.iManPosition, iManVelocity := "ServoV90_A3".In.iManVelocity, iMode := 2, iAListNumber := "ServoV90_A3".Auto.Index, iMListNumber := "ServoV90_A3".Manual.Index, iHWIDSTW := "OP10_382A1~Drive_object~Telegram", iHWIDZSW := "OP10_382A1~Drive_object~Telegram", iHardwareId := "OP10_382A1~Drive_object~Telegram", iHomeSwitch := "iC-GlueServoHomePos", iIndexTableON := FALSE, Position_sensor_1 :=, Position_sensor_2 :=, Position_sensor_3 :=, Position_sensor_4 :=, "Type" :=, TeachMode_Active := "DB_PARAMETERS_TEACH".HMI_PAGE_CONTROL.TEACH_MODE_ACTIVE, ioManEnale := "ServoV90_A3".IO.ioManEnale, ioAutoEnale := "ServoV90_A3".IO.ioAutoEnale, ioHome := "ServoV90_A3".IO.ioAutoHome, ioHomeWrite :=, ioBusy :=, ioDone :=, oReady => "ServoV90_A3".Out.oReady, oWarning => "ServoV90_A3".Out.oWarning, oError => "ServoV90_A3".Out.oError, oInterlock => "ServoV90_A3".Out.oInterlock, oServoEnable => "ServoV90_A3".Out.oServoEnable, oRunning => "ServoV90_A3".Out.oRunning, oHoming => "ServoV90_A3".Out.oHoming, oHomeRef => "ServoV90_A3".Out.oHomeRef, oServoPosOK => "ServoV90_A3".Out.oServoPosOK, oErrorCode => "ServoV90_A3".Out.oErrorCode, oStatus => "ServoV90_A3".Out.oStatus, oActPosition => "ServoV90_A3".Out.oActPosition, oTargetPos =>, oPosOK => "ServoV90_A3".PositionOk, oDisable =>, oSensorInPos =>)
   END_RUNG
   RUNG wire#powerrail
      { S7_Templates := "SrcType := Int" } EQ_Contact(in1 := "ST10_PM".Num[7].StepNum, in2 := 288)
   END_RUNG wire#w1
   RUNG wire#powerrail
      { S7_Templates := "SrcType := Int" } EQ_Contact(in1 := "ST10_PM".Num[6].StepNum, in2 := 422)
      I_Contact( "iC-GlueServoHomePos" )
   END_RUNG wire#w1
   // the same network as SCL:
   #Servo_382A1(iSysRun := "Station_Sys".Status.Run,   // "fbV90Ctrl"
                iReset := "Station_Sys".Cmd.Reset,
                iEstop := "Station_Sys".Status.EStopOK,
                iAuto := "Station_Sys".Auto.Mode,
                iManual := "Station_Sys".Manual.Mode,
                iConnect := true,
                iInterlock := "ServoV90_A3".In.iInterlock,
                "iManJog+" := "ServoV90_A3".In."iManJog+",
                "iManJog-" := "ServoV90_A3".In."iManJog-",
                iManStart := "ServoV90_A3".In.iManStart,
                iManListStart := "ServoV90_A3".In.iManListStart,
                iAutoStart := "ServoV90_A3".In.iAutoStart,
                iRunningTimeout := t#40s,
                iHomingTimeout := t#10s,
                iAutoPosition := "ServoV90_A3".Auto.Pos["ServoV90_A3".Auto.Index].Pos,
                iAutoVelocity := "ServoV90_A3".Auto.Pos["ServoV90_A3".Auto.Index].Vel,
                iManListPosition := "ServoV90_A3".Manual.Pos["ServoV90_A3".Manual.Index].Pos,
                iManListVelocity := "ServoV90_A3".Manual.Pos["ServoV90_A3".Manual.Index].Vel,
                iManPosition := "ServoV90_A3".In.iManPosition,
                iManVelocity := "ServoV90_A3".In.iManVelocity,
                iMode := 2,
                iAListNumber := "ServoV90_A3".Auto.Index,
                iMListNumber := "ServoV90_A3".Manual.Index,
                iHWIDSTW := "OP10_382A1~Drive_object~Telegram",
                iHWIDZSW := "OP10_382A1~Drive_object~Telegram",
                iHardwareId := "OP10_382A1~Drive_object~Telegram",
                iSpecJog := ("ST10_PM".Num[7].StepNum = 288) OR (("ST10_PM".Num[6].StepNum = 422) AND NOT "iC-GlueServoHomePos"),
                iHomeSwitch := "iC-GlueServoHomePos",
                iIndexTableON := FALSE,
                TeachMode_Active := "DB_PARAMETERS_TEACH".HMI_PAGE_CONTROL.TEACH_MODE_ACTIVE,
                ioManEnale := "ServoV90_A3".IO.ioManEnale,
                ioAutoEnale := "ServoV90_A3".IO.ioAutoEnale,
                ioHome := "ServoV90_A3".IO.ioAutoHome,
                oReady => "ServoV90_A3".Out.oReady,
                oWarning => "ServoV90_A3".Out.oWarning,
                oError => "ServoV90_A3".Out.oError,
                oInterlock => "ServoV90_A3".Out.oInterlock,
                oServoEnable => "ServoV90_A3".Out.oServoEnable,
                oRunning => "ServoV90_A3".Out.oRunning,
                oHoming => "ServoV90_A3".Out.oHoming,
                oHomeRef => "ServoV90_A3".Out.oHomeRef,
                oServoPosOK => "ServoV90_A3".Out.oServoPosOK,
                oErrorCode => "ServoV90_A3".Out.oErrorCode,
                oStatus => "ServoV90_A3".Out.oStatus,
                oActPosition => "ServoV90_A3".Out.oActPosition,
                oPosOK => "ServoV90_A3".PositionOk);
END_REGION

REGION Network 31: 复位启动
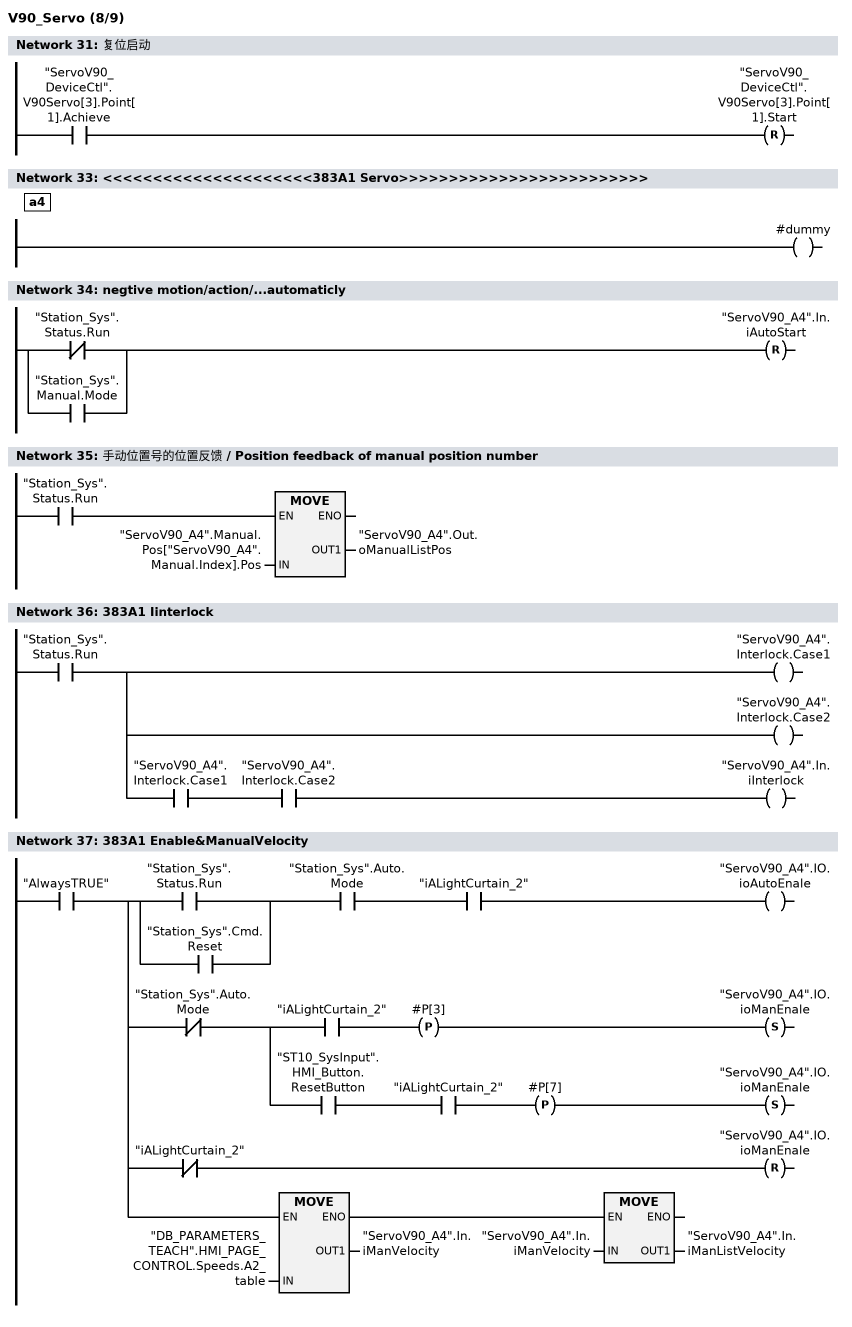
   RUNG wire#powerrail
      Contact( "ServoV90_DeviceCtl".V90Servo[3].Point[1].Achieve )
      R_Coil( "ServoV90_DeviceCtl".V90Servo[3].Point[1].Start )
   END_RUNG
   // the same network as SCL:
   IF "ServoV90_DeviceCtl".V90Servo[3].Point[1].Achieve THEN
       "ServoV90_DeviceCtl".V90Servo[3].Point[1].Start := FALSE;
   END_IF;
END_REGION

REGION Network 32 (SCL): 故障显示 / Fault indication
   //"ST70_DeviceError".Servo2.ServoDriverError := "ServoV90_A3".Out.oError;
END_REGION

REGION Network 33: <<<<<<<<<<<<<<<<<<<<<383A1 Servo>>>>>>>>>>>>>>>>>>>>>>>>>
   Label( a4 )
   RUNG wire#powerrail
      Coil( #dummy )
   END_RUNG
   // the same network as SCL:
   a4:
   #dummy := TRUE;
END_REGION

REGION Network 34: negtive motion/action/...automaticly
   RUNG wire#powerrail
      I_Contact( "Station_Sys".Status.Run )
      wire#w1
      R_Coil( "ServoV90_A4".In.iAutoStart )
   END_RUNG
   RUNG wire#powerrail
      Contact( "Station_Sys".Manual.Mode )
   END_RUNG wire#w1
   // the same network as SCL:
   IF NOT "Station_Sys".Status.Run OR "Station_Sys".Manual.Mode THEN
       "ServoV90_A4".In.iAutoStart := FALSE;
   END_IF;
END_REGION

REGION Network 35: 手动位置号的位置反馈 / Position feedback of manual position number
   RUNG wire#powerrail
      Contact( "Station_Sys".Status.Run )
      Move(in := "ServoV90_A4".Manual.Pos["ServoV90_A4".Manual.Index].Pos, out1 => "ServoV90_A4".Out.oManualListPos)
   END_RUNG
   // the same network as SCL:
   IF "Station_Sys".Status.Run THEN
       "ServoV90_A4".Out.oManualListPos := "ServoV90_A4".Manual.Pos["ServoV90_A4".Manual.Index].Pos;
   END_IF;
END_REGION

REGION Network 36: 383A1 Iinterlock
   RUNG wire#powerrail
      Contact( "Station_Sys".Status.Run )
      wire#w1
      Coil( "ServoV90_A4".Interlock.Case1 )
   END_RUNG
   RUNG wire#w1
      Coil( "ServoV90_A4".Interlock.Case2 )
   END_RUNG
   RUNG wire#w1
      Contact( "ServoV90_A4".Interlock.Case1 )
      Contact( "ServoV90_A4".Interlock.Case2 )
      Coil( "ServoV90_A4".In.iInterlock )
   END_RUNG
   // the same network as SCL:
   "ServoV90_A4".Interlock.Case1 := "Station_Sys".Status.Run;
   "ServoV90_A4".Interlock.Case2 := "Station_Sys".Status.Run;
   "ServoV90_A4".In.iInterlock := "Station_Sys".Status.Run AND "ServoV90_A4".Interlock.Case1 AND "ServoV90_A4".Interlock.Case2;
END_REGION

REGION Network 37: 383A1 Enable&ManualVelocity
   RUNG wire#powerrail
      Contact( "AlwaysTRUE" )
      wire#w1
      Contact( "Station_Sys".Status.Run )
      wire#w2
      Contact( "Station_Sys".Auto.Mode )
      Contact( "iALightCurtain_2" )
      Coil( "ServoV90_A4".IO.ioAutoEnale )
   END_RUNG
   RUNG wire#w1
      Contact( "Station_Sys".Cmd.Reset )
   END_RUNG wire#w2
   RUNG wire#w1
      I_Contact( "Station_Sys".Auto.Mode )
      wire#w3
      Contact( "iALightCurtain_2" )
      P_Trig( #P[3] )
      S_Coil( "ServoV90_A4".IO.ioManEnale )
   END_RUNG
   RUNG wire#w3
      Contact( "ST10_SysInput".HMI_Button.ResetButton )
      Contact( "iALightCurtain_2" )
      P_Trig( #P[7] )
      S_Coil( "ServoV90_A4".IO.ioManEnale )
   END_RUNG
   RUNG wire#w1
      I_Contact( "iALightCurtain_2" )
      R_Coil( "ServoV90_A4".IO.ioManEnale )
   END_RUNG
   RUNG wire#w1
      Move(in := "DB_PARAMETERS_TEACH".HMI_PAGE_CONTROL.Speeds.A2_table, out1 => "ServoV90_A4".In.iManVelocity)
      Move(in := "ServoV90_A4".In.iManVelocity, out1 => "ServoV90_A4".In.iManListVelocity)
   END_RUNG
   // the same network as SCL:
   "ServoV90_A4".IO.ioAutoEnale := "AlwaysTRUE" AND ("Station_Sys".Status.Run OR "Station_Sys".Cmd.Reset) AND "Station_Sys".Auto.Mode AND "iALightCurtain_2";
   #_w1 := "AlwaysTRUE" AND NOT "Station_Sys".Auto.Mode;
   #_w2 := #_w1 AND "iALightCurtain_2";
   #_w3 := #_w2 AND NOT #P[3];   // rising edge
   #P[3] := #_w2;
   IF #_w3 THEN "ServoV90_A4".IO.ioManEnale := TRUE; END_IF;
   #_w4 := #_w1 AND "ST10_SysInput".HMI_Button.ResetButton AND "iALightCurtain_2";
   #_w5 := #_w4 AND NOT #P[7];   // rising edge
   #P[7] := #_w4;
   IF #_w5 THEN "ServoV90_A4".IO.ioManEnale := TRUE; END_IF;
   IF "AlwaysTRUE" AND NOT "iALightCurtain_2" THEN "ServoV90_A4".IO.ioManEnale := FALSE; END_IF;
   IF "AlwaysTRUE" THEN
       "ServoV90_A4".In.iManVelocity := "DB_PARAMETERS_TEACH".HMI_PAGE_CONTROL.Speeds.A2_table;
       "ServoV90_A4".In.iManListVelocity := "ServoV90_A4".In.iManVelocity;
   END_IF;
END_REGION

REGION Network 38 (SCL): 383A1 RecipePosition
   IF "Station_Sys".Status.Run THEN
       "ServoV90_A4".Manual.Pos[1].Pos := "ServoV90_A4".Auto.Pos[1].Pos := REAL_TO_DINT("Parameter".AxisRun.Axis[4].Pos1.Position*1000);
       "ServoV90_A4".Manual.Pos[1].Vel := "ServoV90_A4".Auto.Pos[1].Vel := "Parameter".AxisRun.Axis[4].Pos1.Speed;

       "ServoV90_A4".Manual.Pos[2].Pos := "ServoV90_A4".Auto.Pos[2].Pos := REAL_TO_DINT("Parameter".AxisRun.Axis[4].Pos2.Position*1000);
       "ServoV90_A4".Manual.Pos[2].Vel := "ServoV90_A4".Auto.Pos[2].Vel := "Parameter".AxisRun.Axis[4].Pos2.Speed;

       "ServoV90_A4".Manual.Pos[3].Pos := "ServoV90_A4".Auto.Pos[3].Pos := REAL_TO_DINT("Parameter".AxisRun.Axis[4].Pos3.Position*1000);
       "ServoV90_A4".Manual.Pos[3].Vel := "ServoV90_A4".Auto.Pos[3].Vel := "Parameter".AxisRun.Axis[4].Pos3.Speed;

       "ServoV90_A4".Manual.Pos[4].Pos := "ServoV90_A4".Auto.Pos[4].Pos := REAL_TO_DINT("Parameter".AxisRun.Axis[4].Pos4.Position*1000);
       "ServoV90_A4".Manual.Pos[4].Vel := "ServoV90_A4".Auto.Pos[4].Vel := "Parameter".AxisRun.Axis[4].Pos4.Speed;

       "ServoV90_A4".Manual.Pos[5].Pos := "ServoV90_A4".Auto.Pos[5].Pos := REAL_TO_DINT("Parameter".AxisRun.Axis[4].Pos5.Position*1000);
       "ServoV90_A4".Manual.Pos[5].Vel := "ServoV90_A4".Auto.Pos[5].Vel := "Parameter".AxisRun.Axis[4].Pos5.Speed;

       "ServoV90_A4".Manual.Pos[6].Pos := "ServoV90_A4".Auto.Pos[6].Pos := REAL_TO_DINT("Parameter".AxisRun.Axis[4].Pos6.Position*1000);
       "ServoV90_A4".Manual.Pos[6].Vel := "ServoV90_A4".Auto.Pos[6].Vel := "Parameter".AxisRun.Axis[4].Pos6.Speed;

       "ServoV90_A4".Manual.Pos[7].Pos := "ServoV90_A4".Auto.Pos[7].Pos := REAL_TO_DINT("Parameter".AxisRun.Axis[4].Pos7.Position*1000);
       "ServoV90_A4".Manual.Pos[7].Vel := "ServoV90_A4".Auto.Pos[7].Vel := "Parameter".AxisRun.Axis[4].Pos7.Speed;

       "ServoV90_A4".Manual.Pos[8].Pos := "ServoV90_A4".Auto.Pos[8].Pos := REAL_TO_DINT("Parameter".AxisRun.Axis[4].Pos8.Position*1000);
       "ServoV90_A4".Manual.Pos[8].Vel := "ServoV90_A4".Auto.Pos[8].Vel := "Parameter".AxisRun.Axis[4].Pos8.Speed;

       "ServoV90_A4".Manual.Pos[9].Pos := "ServoV90_A4".Auto.Pos[9].Pos := REAL_TO_DINT("Parameter".AxisRun.Axis[4].Pos9.Position*1000);
       "ServoV90_A4".Manual.Pos[9].Vel := "ServoV90_A4".Auto.Pos[9].Vel := "Parameter".AxisRun.Axis[4].Pos9.Speed;

       "ServoV90_A4".Manual.Pos[10].Pos := "ServoV90_A4".Auto.Pos[10].Pos := REAL_TO_DINT("Parameter".AxisRun.Axis[4].Pos10.Position*1000);
       "ServoV90_A4".Manual.Pos[10].Vel := "ServoV90_A4".Auto.Pos[10].Vel := "Parameter".AxisRun.Axis[4].Pos10.Speed;
   END_IF;
END_REGION

REGION Network 39: 383A1 FB
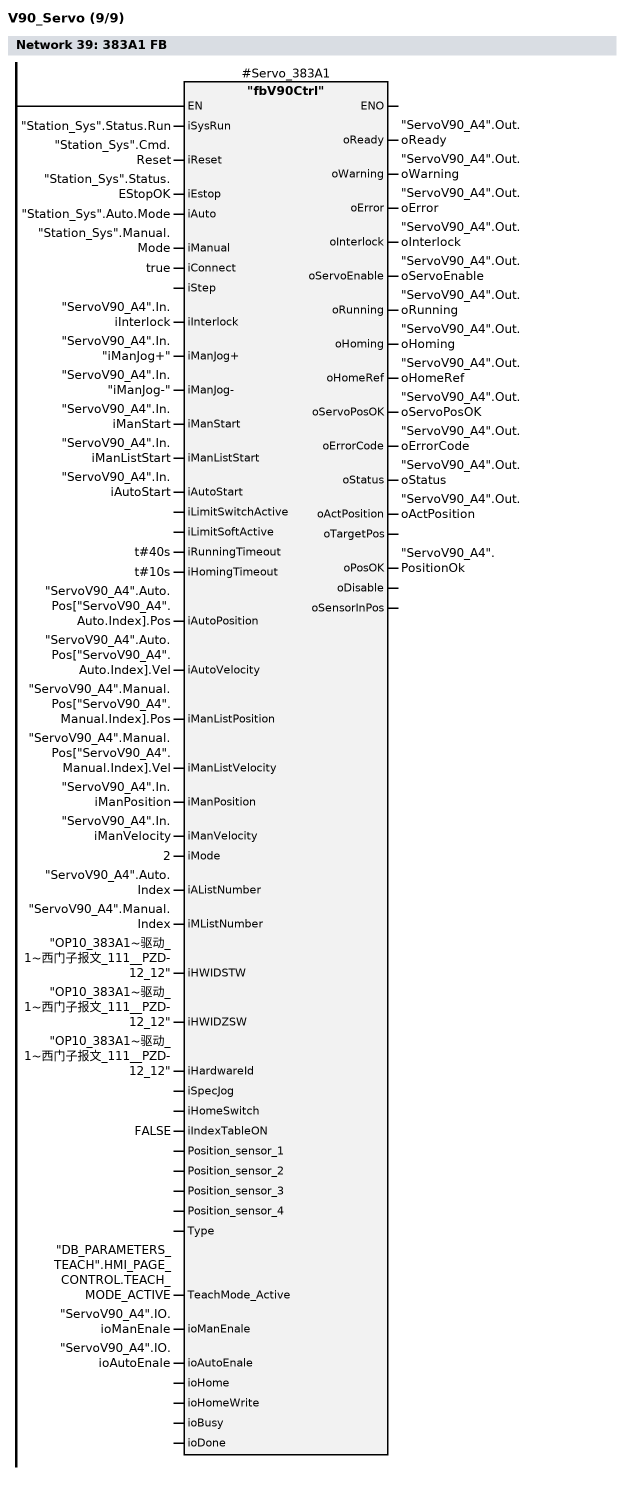
   RUNG wire#powerrail
      #Servo_383A1(iSysRun := "Station_Sys".Status.Run, iReset := "Station_Sys".Cmd.Reset, iEstop := "Station_Sys".Status.EStopOK, iAuto := "Station_Sys".Auto.Mode, iManual := "Station_Sys".Manual.Mode, iConnect := true, iStep :=, iInterlock := "ServoV90_A4".In.iInterlock, "iManJog+" := "ServoV90_A4".In."iManJog+", "iManJog-" := "ServoV90_A4".In."iManJog-", iManStart := "ServoV90_A4".In.iManStart, iManListStart := "ServoV90_A4".In.iManListStart, iAutoStart := "ServoV90_A4".In.iAutoStart, iLimitSwitchActive :=, iLimitSoftActive :=, iRunningTimeout := t#40s, iHomingTimeout := t#10s, iAutoPosition := "ServoV90_A4".Auto.Pos["ServoV90_A4".Auto.Index].Pos, iAutoVelocity := "ServoV90_A4".Auto.Pos["ServoV90_A4".Auto.Index].Vel, iManListPosition := "ServoV90_A4".Manual.Pos["ServoV90_A4".Manual.Index].Pos, iManListVelocity := "ServoV90_A4".Manual.Pos["ServoV90_A4".Manual.Index].Vel, iManPosition := "ServoV90_A4".In.iManPosition, iManVelocity := "ServoV90_A4".In.iManVelocity, iMode := 2, iAListNumber := "ServoV90_A4".Auto.Index, iMListNumber := "ServoV90_A4".Manual.Index, iHWIDSTW := "OP10_383A1~驱动_1~西门子报文_111__PZD-12_12", iHWIDZSW := "OP10_383A1~驱动_1~西门子报文_111__PZD-12_12", iHardwareId := "OP10_383A1~驱动_1~西门子报文_111__PZD-12_12", iSpecJog :=, iHomeSwitch :=, iIndexTableON := FALSE, Position_sensor_1 :=, Position_sensor_2 :=, Position_sensor_3 :=, Position_sensor_4 :=, "Type" :=, TeachMode_Active := "DB_PARAMETERS_TEACH".HMI_PAGE_CONTROL.TEACH_MODE_ACTIVE, ioManEnale := "ServoV90_A4".IO.ioManEnale, ioAutoEnale := "ServoV90_A4".IO.ioAutoEnale, ioHome :=, ioHomeWrite :=, ioBusy :=, ioDone :=, oReady => "ServoV90_A4".Out.oReady, oWarning => "ServoV90_A4".Out.oWarning, oError => "ServoV90_A4".Out.oError, oInterlock => "ServoV90_A4".Out.oInterlock, oServoEnable => "ServoV90_A4".Out.oServoEnable, oRunning => "ServoV90_A4".Out.oRunning, oHoming => "ServoV90_A4".Out.oHoming, oHomeRef => "ServoV90_A4".Out.oHomeRef, oServoPosOK => "ServoV90_A4".Out.oServoPosOK, oErrorCode => "ServoV90_A4".Out.oErrorCode, oStatus => "ServoV90_A4".Out.oStatus, oActPosition => "ServoV90_A4".Out.oActPosition, oTargetPos =>, oPosOK => "ServoV90_A4".PositionOk, oDisable =>, oSensorInPos =>)
   END_RUNG
   // the same network as SCL:
   #Servo_383A1(iSysRun := "Station_Sys".Status.Run,   // "fbV90Ctrl"
                iReset := "Station_Sys".Cmd.Reset,
                iEstop := "Station_Sys".Status.EStopOK,
                iAuto := "Station_Sys".Auto.Mode,
                iManual := "Station_Sys".Manual.Mode,
                iConnect := true,
                iInterlock := "ServoV90_A4".In.iInterlock,
                "iManJog+" := "ServoV90_A4".In."iManJog+",
                "iManJog-" := "ServoV90_A4".In."iManJog-",
                iManStart := "ServoV90_A4".In.iManStart,
                iManListStart := "ServoV90_A4".In.iManListStart,
                iAutoStart := "ServoV90_A4".In.iAutoStart,
                iRunningTimeout := t#40s,
                iHomingTimeout := t#10s,
                iAutoPosition := "ServoV90_A4".Auto.Pos["ServoV90_A4".Auto.Index].Pos,
                iAutoVelocity := "ServoV90_A4".Auto.Pos["ServoV90_A4".Auto.Index].Vel,
                iManListPosition := "ServoV90_A4".Manual.Pos["ServoV90_A4".Manual.Index].Pos,
                iManListVelocity := "ServoV90_A4".Manual.Pos["ServoV90_A4".Manual.Index].Vel,
                iManPosition := "ServoV90_A4".In.iManPosition,
                iManVelocity := "ServoV90_A4".In.iManVelocity,
                iMode := 2,
                iAListNumber := "ServoV90_A4".Auto.Index,
                iMListNumber := "ServoV90_A4".Manual.Index,
                iHWIDSTW := "OP10_383A1~驱动_1~西门子报文_111__PZD-12_12",
                iHWIDZSW := "OP10_383A1~驱动_1~西门子报文_111__PZD-12_12",
                iHardwareId := "OP10_383A1~驱动_1~西门子报文_111__PZD-12_12",
                iIndexTableON := FALSE,
                TeachMode_Active := "DB_PARAMETERS_TEACH".HMI_PAGE_CONTROL.TEACH_MODE_ACTIVE,
                ioManEnale := "ServoV90_A4".IO.ioManEnale,
                ioAutoEnale := "ServoV90_A4".IO.ioAutoEnale,
                oReady => "ServoV90_A4".Out.oReady,
                oWarning => "ServoV90_A4".Out.oWarning,
                oError => "ServoV90_A4".Out.oError,
                oInterlock => "ServoV90_A4".Out.oInterlock,
                oServoEnable => "ServoV90_A4".Out.oServoEnable,
                oRunning => "ServoV90_A4".Out.oRunning,
                oHoming => "ServoV90_A4".Out.oHoming,
                oHomeRef => "ServoV90_A4".Out.oHomeRef,
                oServoPosOK => "ServoV90_A4".Out.oServoPosOK,
                oErrorCode => "ServoV90_A4".Out.oErrorCode,
                oStatus => "ServoV90_A4".Out.oStatus,
                oActPosition => "ServoV90_A4".Out.oActPosition,
                oPosOK => "ServoV90_A4".PositionOk);
END_REGION

REGION Network 40 (SCL): 故障显示 / Fault indication
   //"ST70_DeviceError".Servo2.ServoDriverError := "ServoV90_A4".Out.oError;
END_REGION

REGION Network 41: *********************************伺服位置判断**********************************************
END_REGION

REGION Network 42 (SCL): 伺服位置判断 / Servo position judgment
   FOR "ServoV90_DeviceCtl".V90Servo[1].i := 1 TO 12 BY 1 DO
       "ServoV90_DeviceCtl".V90Servo[1].Pos.List["ServoV90_DeviceCtl".V90Servo[1].i].Pos := "ServoV90_A1".Auto.Pos["ServoV90_DeviceCtl".V90Servo[1].i].Pos;
       "ServoV90_DeviceCtl".V90Servo[1].Pos.List["ServoV90_DeviceCtl".V90Servo[1].i].Vel := "ServoV90_A1".Auto.Pos["ServoV90_DeviceCtl".V90Servo[1].i].Vel;

       "ServoV90_DeviceCtl".V90Servo[2].Pos.List["ServoV90_DeviceCtl".V90Servo[1].i].Pos := "ServoV90_A2".Auto.Pos["ServoV90_DeviceCtl".V90Servo[1].i].Pos;
       "ServoV90_DeviceCtl".V90Servo[2].Pos.List["ServoV90_DeviceCtl".V90Servo[1].i].Vel := "ServoV90_A2".Auto.Pos["ServoV90_DeviceCtl".V90Servo[1].i].Vel;

       "ServoV90_DeviceCtl".V90Servo[3].Pos.List["ServoV90_DeviceCtl".V90Servo[1].i].Pos := "ServoV90_A3".Auto.Pos["ServoV90_DeviceCtl".V90Servo[1].i].Pos;
       "ServoV90_DeviceCtl".V90Servo[3].Pos.List["ServoV90_DeviceCtl".V90Servo[1].i].Vel := "ServoV90_A3".Auto.Pos["ServoV90_DeviceCtl".V90Servo[1].i].Vel;

       "ServoV90_DeviceCtl".V90Servo[4].Pos.List["ServoV90_DeviceCtl".V90Servo[1].i].Pos := "ServoV90_A4".Auto.Pos["ServoV90_DeviceCtl".V90Servo[1].i].Pos;
       "ServoV90_DeviceCtl".V90Servo[4].Pos.List["ServoV90_DeviceCtl".V90Servo[1].i].Vel := "ServoV90_A4".Auto.Pos["ServoV90_DeviceCtl".V90Servo[1].i].Vel;

   END_FOR;

   (******************************************************* SV1 ********************************************************************)   
   //伺服位置判断
   #"Servo1"(iRef_Homed :=   "ServoV90_A1".Out.oHomeRef,
                             iStandstill := FALSE,
                             iReset := "Station_Sys".Cmd.Reset,
                             interlcok:="ServoV90_A1".In.iInterlock,
                             "iActual Posi" :="ServoV90_A1".Out.oActPosition,
                             "iTol+" := 50,
                             "iTol-" := 50,
                             iStartTon := T#100mS,
                             ioPoint:="ServoV90_DeviceCtl".V90Servo[1].Point,
                             oStartPos => #Sevro1StartList,
                             ioList := "ServoV90_DeviceCtl".V90Servo[1].Pos,
                             ioPosNumberSelect := "ServoV90_DeviceCtl".V90Servo[1].nPositionListNo);

   IF "ServoV90_DeviceCtl".V90Servo[1].nPositionListNo = 0 THEN
      "ServoV90_DeviceCtl".V90Servo[1].nPositionListNo:= 1 ;
   END_IF;

    //伺服位置号给定
                   // IF NOT "D-2 ModuleD-2 横向抓取移栽/拍照/旋转_IDB".伺服到下料位.X THEN
                   //     "ServoV90_A1".Auto.Index := "ServoV90_DeviceCtl".V90Servo[1].nPositionListNo;
                   // END_IF;

                  "ServoV90_A1".Auto.Index := "ServoV90_DeviceCtl".V90Servo[1].nPositionListNo;

   //伺服启动
                   "ServoV90_A1".In.iAutoStart := #Sevro1StartList;


   (******************************************************* SV2 ********************************************************************)                
   //伺服位置判断
   #"Servo2"(iRef_Homed := "ServoV90_A2".Out.oHomeRef,
             iStandstill := FALSE,
             iReset := "Station_Sys".Cmd.Reset,
             interlcok := "ServoV90_A2".In.iInterlock,
             "iActual Posi" := "ServoV90_A2".Out.oActPosition,
             "iTol+" := 50,
             "iTol-" := 50,
             iStartTon := T#100mS,
             ioPoint := "ServoV90_DeviceCtl".V90Servo[2].Point,
             oStartPos => #Sevro2StartList,
             ioList := "ServoV90_DeviceCtl".V90Servo[2].Pos,
             ioPosNumberSelect := "ServoV90_DeviceCtl".V90Servo[2].nPositionListNo);

   IF "ServoV90_DeviceCtl".V90Servo[2].nPositionListNo = 0 THEN
       "ServoV90_DeviceCtl".V90Servo[2].nPositionListNo := 1;
   END_IF;

   //伺服位置号给定
   // IF NOT "D-3 ModuleD-3从转台下料到托盘移栽机构_IDB".移栽伺服到取料位1.X THEN
   //     "ServoV90_A2".Auto.Index := "ServoV90_DeviceCtl".CMMTServo[2].nPositionListNo;
   // END_IF;

   "ServoV90_A2".Auto.Index := "ServoV90_DeviceCtl".V90Servo[2].nPositionListNo;

   //伺服启动
   "ServoV90_A2".In.iAutoStart := #Sevro2StartList;


   (******************************************************* SV3 ********************************************************************)
   //伺服位置判断
   #"Servo3"(iRef_Homed := "ServoV90_A3".Out.oHomeRef,
             iStandstill := FALSE,
             iReset := "Station_Sys".Cmd.Reset,
             interlcok := "ServoV90_A3".In.iInterlock,
             "iActual Posi" := "ServoV90_A3".Out.oActPosition,
             "iTol+" := 50,
             "iTol-" := 50,
             iStartTon := T#100mS,
             ioPoint := "ServoV90_DeviceCtl".V90Servo[3].Point,
             oStartPos => #Sevro3StartList,
             ioList := "ServoV90_DeviceCtl".V90Servo[3].Pos,
             ioPosNumberSelect := "ServoV90_DeviceCtl".V90Servo[3].nPositionListNo);

   IF "ServoV90_DeviceCtl".V90Servo[3].nPositionListNo = 0 THEN
       "ServoV90_DeviceCtl".V90Servo[3].nPositionListNo := 1;
   END_IF;
   //伺服位置号给定
   // IF NOT "D-3 ModuleD-3从转台下料到托盘移栽机构_IDB".移栽伺服到取料位1.X THEN
   //     "ServoV90_A2".Auto.Index := "ServoV90_DeviceCtl".V90Servo[2].nPositionListNo;
   // END_IF;

   "ServoV90_A3".Auto.Index := "ServoV90_DeviceCtl".V90Servo[3].nPositionListNo;

   //伺服启动
   "ServoV90_A3".In.iAutoStart := #Sevro3StartList;


   (******************************************************* SV4 ********************************************************************)
   //伺服位置判断
   #"Servo4"(iRef_Homed := "ServoV90_A4".Out.oHomeRef,
             iStandstill := FALSE,
             iReset := "Station_Sys".Cmd.Reset,
             interlcok := "ServoV90_A4".In.iInterlock,
             "iActual Posi" := "ServoV90_A4".Out.oActPosition,
             "iTol+" := 50,
             "iTol-" := 50,
             iStartTon := T#100mS,
             ioPoint := "ServoV90_DeviceCtl".V90Servo[4].Point,
             oStartPos => #Sevro4StartList,
             ioList := "ServoV90_DeviceCtl".V90Servo[4].Pos,
             ioPosNumberSelect := "ServoV90_DeviceCtl".V90Servo[4].nPositionListNo);

   IF "ServoV90_DeviceCtl".V90Servo[4].nPositionListNo = 0 THEN
       "ServoV90_DeviceCtl".V90Servo[4].nPositionListNo := 1;
   END_IF;

   //伺服位置号给定
   // IF NOT "D-3 ModuleD-3从转台下料到托盘移栽机构_IDB".移栽伺服到取料位1.X THEN
   //     "ServoV90_A2".Auto.Index := "ServoV90_DeviceCtl".V90Servo[2].nPositionListNo;
   // END_IF;

   "ServoV90_A4".Auto.Index := "ServoV90_DeviceCtl".V90Servo[4].nPositionListNo;

   //伺服启动
   "ServoV90_A4".In.iAutoStart := #Sevro4StartList;
END_REGION

REGION Network 43 (SCL): 初始化脉冲 置位手动使能 / The initial pulse set function was manually enabled
   IF "FirstScan" THEN
       "ServoV90_A1".IO.ioManEnale := TRUE;
       "ServoV90_A2".IO.ioManEnale := TRUE;
       "ServoV90_A3".IO.ioManEnale := TRUE;
       "ServoV90_A4".IO.ioManEnale := TRUE;
   END_IF;
END_REGION
END_FUNCTION_BLOCK

FUNCTION_BLOCK "SevroStart&PosCheck"   // FB4073, LAD
{ S7_Optimized_Access := 'TRUE' }
VERSION : 0.1
// stored: AutoNumber false, IsIECCheckEnabled false, IsRetainMemResEnabled false, MemoryReserve 100, SetENOAutomatically false, UDAEnableTagReadback false
   VAR_INPUT
      iRef_Homed { ExternalAccessible := 'False'; ExternalVisible := 'False'; ExternalWritable := 'False'} : Bool;
      iStandstill { ExternalAccessible := 'False'; ExternalVisible := 'False'; ExternalWritable := 'False'} : Bool;
      iReset : Bool;
      interlcok : Bool;   // 启动互锁
      "iActual Posi" { ExternalAccessible := 'False'; ExternalVisible := 'False'; ExternalWritable := 'False'} : DInt;
      "iTol+" { ExternalAccessible := 'False'; ExternalVisible := 'False'; ExternalWritable := 'False'} : DInt;
      "iTol-" { ExternalAccessible := 'False'; ExternalVisible := 'False'; ExternalWritable := 'False'} : DInt;
      iStartTon : Time := T#200ms;   // 启动延迟
   END_VAR
   VAR_OUTPUT
      oStartPos : Bool;   // 启动
      DoublePosError : Bool;   // 多位置触发
   END_VAR
   VAR_IN_OUT
      ioPoint : Array[0..39] of Struct
         Start : Bool;
         Achieve : Bool;
      END_STRUCT;
      ioList : "PosList";
      ioPosNumberSelect : Int;   // 位置启动
   END_VAR
   VAR
      TON : Array[0..1] of TON_TIME;
      StartCount { S7_SetPoint := 'True'} : Int;   // 启动计数
   END_VAR
   VAR_TEMP
      "Actual Posi+Tol" : DInt;
      "Actual Posi-Tol" : DInt;
      Index : Array[0..7] of Int;   // 位置启动
      PosStart : Bool;
   END_VAR
   VAR_TEMP   // added for the SCL form of the ladder/FBD networks
      _w1 : Bool;
   END_VAR
BEGIN

REGION Network 1 (SCL): 检查当前启动位置号
   #Index[1] := 0;
   #PosStart := false;
   FOR #Index[1] := 0 TO 39 DO
       IF #ioPoint[#Index[1]].Start THEN

           #ioPosNumberSelect := #Index[1];//当前启动位置号
           #PosStart := TRUE;
           EXIT;
       END_IF;
   END_FOR;
   #Index[2] := 0;
   #StartCount := 0;
   FOR #Index[2] := 0 TO 39 DO
       IF #ioPoint[#Index[2]].Start THEN

           #StartCount := #StartCount+1;//当前启动位置号


       END_IF;
       IF #Index[2] = 39 THEN

           EXIT;
       END_IF;

   END_FOR;
END_REGION

REGION Network 2: 位置给定
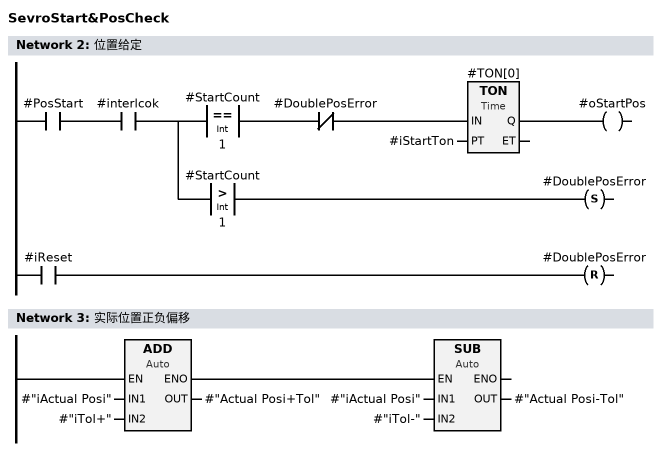
   RUNG wire#powerrail
      Contact( #PosStart )
      Contact( #interlcok )
      wire#w1
      { S7_Templates := "SrcType := Int" } EQ_Contact(in1 := #StartCount, in2 := 1)
      I_Contact( #DoublePosError )
      { S7_Templates := "time_type := Time" } #TON[0].TON(pt := #iStartTon, et =>)
      Coil( #oStartPos )
   END_RUNG
   RUNG wire#w1
      { S7_Templates := "SrcType := Int" } GT_Contact(in1 := #StartCount, in2 := 1)
      S_Coil( #DoublePosError )
   END_RUNG
   RUNG wire#powerrail
      Contact( #iReset )
      R_Coil( #DoublePosError )
   END_RUNG
   // the same network as SCL:
   #_w1 := #PosStart AND #interlcok;
   #TON[0].TON(IN := #_w1 AND (#StartCount = 1) AND NOT #DoublePosError, PT := #iStartTon);
   #oStartPos := #TON[0].Q;
   IF #_w1 AND (#StartCount > 1) THEN #DoublePosError := TRUE; END_IF;
   IF #iReset THEN #DoublePosError := FALSE; END_IF;
END_REGION

REGION Network 3: 实际位置正负偏移
   RUNG wire#powerrail
      Add(in1 := #"iActual Posi", in2 := #"iTol+", out => #"Actual Posi+Tol")
      Sub(in1 := #"iActual Posi", in2 := #"iTol-", out => #"Actual Posi-Tol")
   END_RUNG
   // the same network as SCL:
   #"Actual Posi+Tol" := #"iActual Posi" + #"iTol+";
   #"Actual Posi-Tol" := #"iActual Posi" - #"iTol-";
END_REGION

REGION Network 4 (SCL): 位置检查


   #Index[3] := 0;
   FOR #Index[3] := 0 TO 39 DO
       IF #ioList.List[ #Index[3]].Pos>= #"Actual Posi-Tol"
           AND #ioList.List[ #Index[3]].Pos<= #"Actual Posi+Tol"
       THEN
         #ioPoint[#Index[3]].Achieve := TRUE;
       ELSE
           #ioPoint[#Index[3]].Achieve := FALSE;
       END_IF;
   END_FOR;
END_REGION
END_FUNCTION_BLOCK

FUNCTION "Motorr" : Void   // FC3100, LAD
{ S7_Optimized_Access := 'TRUE' }
// stored: AutoNumber false, SetENOAutomatically false
   VAR_TEMP   // added for the SCL form of the ladder/FBD networks
      _w1 : Bool;
      _w2 : Bool;
   END_VAR
BEGIN

REGION Network 1: H-shaftLifting_Motor
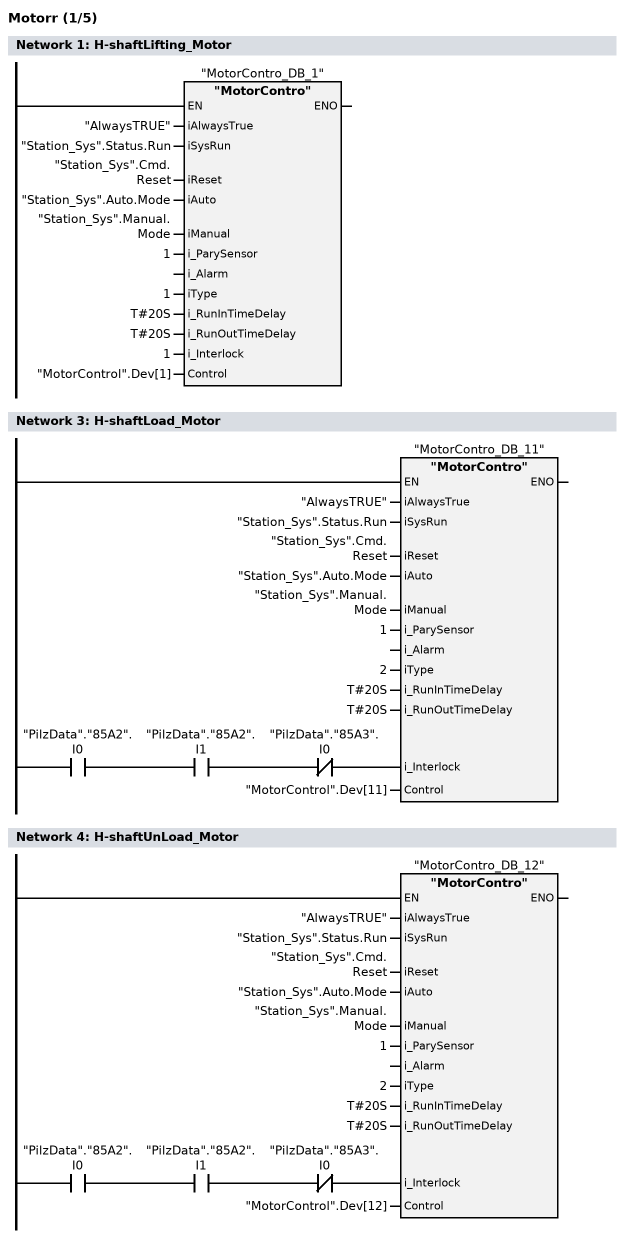
   RUNG wire#powerrail
      "MotorContro_DB_1"(iAlwaysTrue := "AlwaysTRUE", iSysRun := "Station_Sys".Status.Run, iReset := "Station_Sys".Cmd.Reset, iAuto := "Station_Sys".Auto.Mode, iManual := "Station_Sys".Manual.Mode, i_ParySensor := 1, i_Alarm :=, iType := 1, i_RunInTimeDelay := T#20S, i_RunOutTimeDelay := T#20S, i_Interlock := 1, Control := "MotorControl".Dev[1])
   END_RUNG
   // the same network as SCL:
   "MotorContro_DB_1"(iAlwaysTrue := "AlwaysTRUE",   // "MotorContro"
                      iSysRun := "Station_Sys".Status.Run,
                      iReset := "Station_Sys".Cmd.Reset,
                      iAuto := "Station_Sys".Auto.Mode,
                      iManual := "Station_Sys".Manual.Mode,
                      i_ParySensor := 1,
                      iType := 1,
                      i_RunInTimeDelay := T#20S,
                      i_RunOutTimeDelay := T#20S,
                      i_Interlock := 1,
                      Control := "MotorControl".Dev[1]);
END_REGION

REGION Network 2 (SCL): H-shaftLifting_Motor_OutPut
   "oH-shaftLifting_Start" := "MotorControl".Dev[1].OutControl.o_Start;
   "oH-shaftLifting_CCWStart" := "MotorControl".Dev[1].OutControl.o_CCWStart ;
   "oH-shaftLifting_SpeedChange" := "MotorControl".Dev[1].OutControl.o_SpeedChanged;
END_REGION

REGION Network 3: H-shaftLoad_Motor
   RUNG wire#powerrail
      "MotorContro_DB_11"(i_Interlock := wire#w1, iAlwaysTrue := "AlwaysTRUE", iSysRun := "Station_Sys".Status.Run, iReset := "Station_Sys".Cmd.Reset, iAuto := "Station_Sys".Auto.Mode, iManual := "Station_Sys".Manual.Mode, i_ParySensor := 1, i_Alarm :=, iType := 2, i_RunInTimeDelay := T#20S, i_RunOutTimeDelay := T#20S, Control := "MotorControl".Dev[11])
   END_RUNG
   RUNG wire#powerrail
      Contact( "PilzData"."85A2".I0 )
      Contact( "PilzData"."85A2".I1 )
      I_Contact( "PilzData"."85A3".I0 )
   END_RUNG wire#w1
   // the same network as SCL:
   "MotorContro_DB_11"(iAlwaysTrue := "AlwaysTRUE",   // "MotorContro"
                       iSysRun := "Station_Sys".Status.Run,
                       iReset := "Station_Sys".Cmd.Reset,
                       iAuto := "Station_Sys".Auto.Mode,
                       iManual := "Station_Sys".Manual.Mode,
                       i_ParySensor := 1,
                       iType := 2,
                       i_RunInTimeDelay := T#20S,
                       i_RunOutTimeDelay := T#20S,
                       i_Interlock := "PilzData"."85A2".I0 AND "PilzData"."85A2".I1 AND NOT "PilzData"."85A3".I0,
                       Control := "MotorControl".Dev[11]);
END_REGION

REGION Network 4: H-shaftUnLoad_Motor
   RUNG wire#powerrail
      "MotorContro_DB_12"(i_Interlock := wire#w1, iAlwaysTrue := "AlwaysTRUE", iSysRun := "Station_Sys".Status.Run, iReset := "Station_Sys".Cmd.Reset, iAuto := "Station_Sys".Auto.Mode, iManual := "Station_Sys".Manual.Mode, i_ParySensor := 1, i_Alarm :=, iType := 2, i_RunInTimeDelay := T#20S, i_RunOutTimeDelay := T#20S, Control := "MotorControl".Dev[12])
   END_RUNG
   RUNG wire#powerrail
      Contact( "PilzData"."85A2".I0 )
      Contact( "PilzData"."85A2".I1 )
      I_Contact( "PilzData"."85A3".I0 )
   END_RUNG wire#w1
   // the same network as SCL:
   "MotorContro_DB_12"(iAlwaysTrue := "AlwaysTRUE",   // "MotorContro"
                       iSysRun := "Station_Sys".Status.Run,
                       iReset := "Station_Sys".Cmd.Reset,
                       iAuto := "Station_Sys".Auto.Mode,
                       iManual := "Station_Sys".Manual.Mode,
                       i_ParySensor := 1,
                       iType := 2,
                       i_RunInTimeDelay := T#20S,
                       i_RunOutTimeDelay := T#20S,
                       i_Interlock := "PilzData"."85A2".I0 AND "PilzData"."85A2".I1 AND NOT "PilzData"."85A3".I0,
                       Control := "MotorControl".Dev[12]);
END_REGION

REGION Network 5 (SCL): H-shaftLifting_Motor_OutPut / H-shaftLoad_Motor_OutPut
   "oH-shaftLoading_CW" := "MotorControl".Dev[11].OutControl.o_Start;
   "oH-shaftLoading_CCW" := "MotorControl".Dev[11].OutControl.o_CCWStart OR ("Station_Sys".Auto.Mode AND "AutoProcessControl".Global.H.EmptyPallet);

   "oH-shaftTake_CW" := "MotorControl".Dev[12].OutControl.o_Start;
END_REGION

REGION Network 6: Auto MotorStop
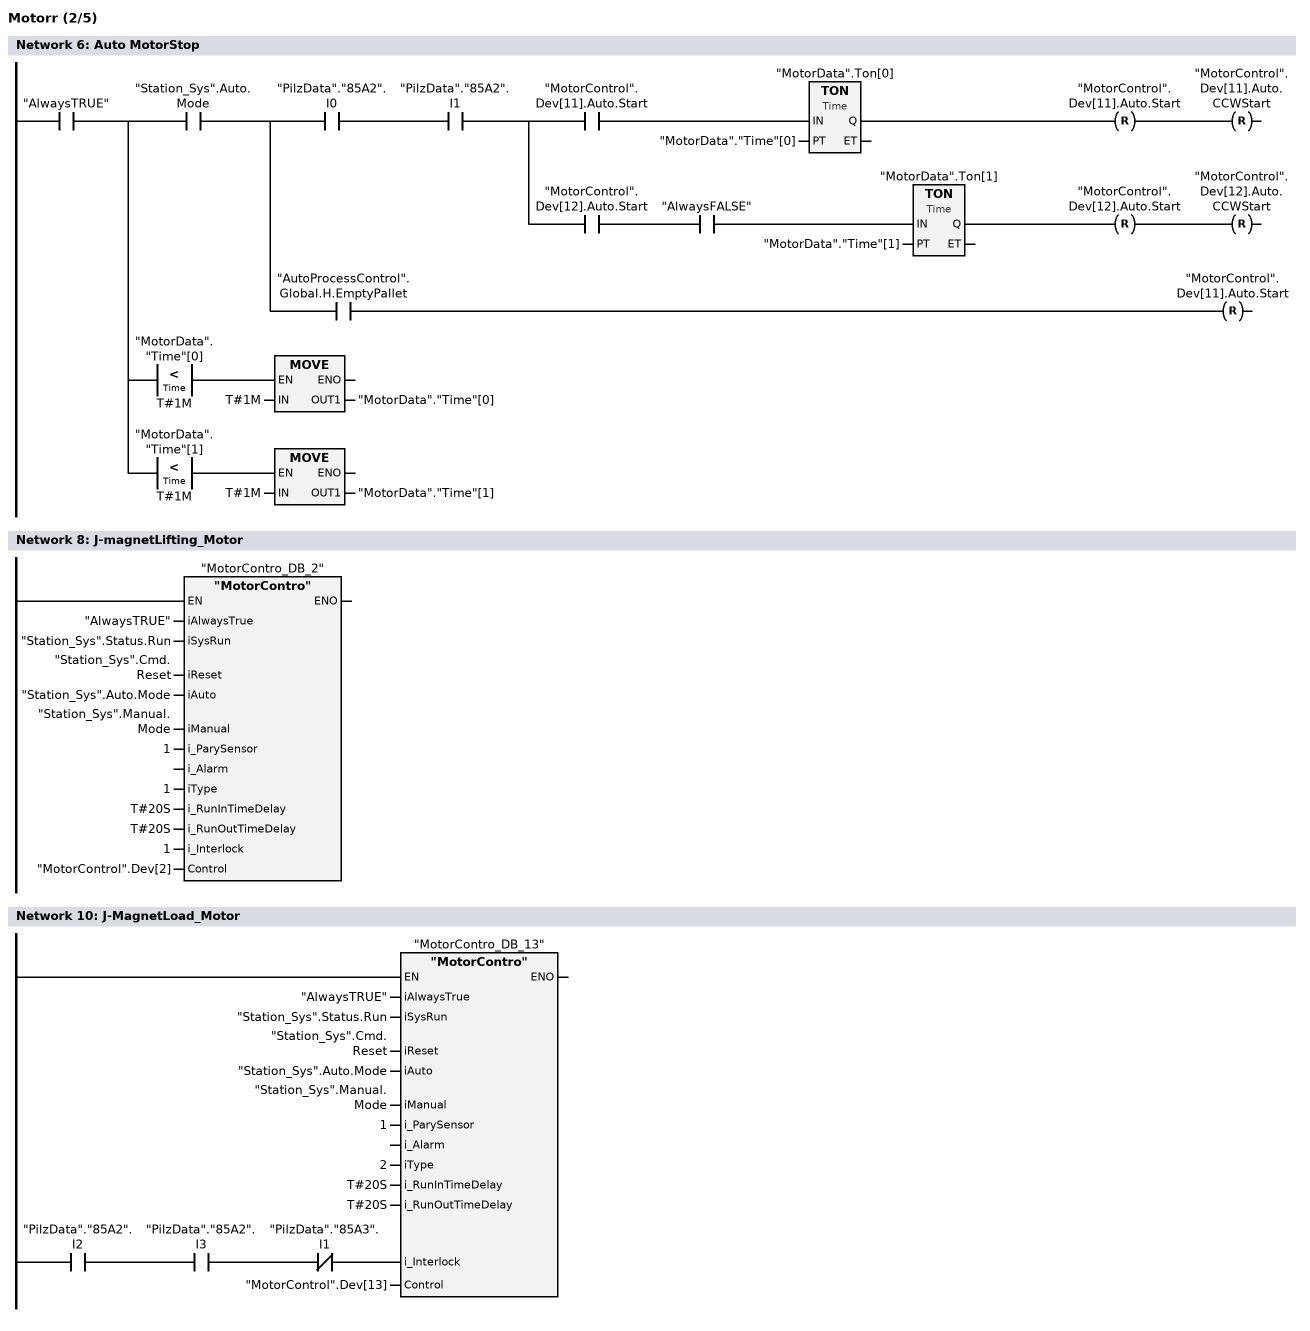
   RUNG wire#powerrail
      Contact( "AlwaysTRUE" )
      wire#w1
      Contact( "Station_Sys".Auto.Mode )
      wire#w2
      Contact( "PilzData"."85A2".I0 )
      Contact( "PilzData"."85A2".I1 )
      wire#w3
      Contact( "MotorControl".Dev[11].Auto.Start )
      { S7_Templates := "time_type := Time" } "MotorData".Ton[0].TON(pt := "MotorData"."Time"[0], et =>)
      R_Coil( "MotorControl".Dev[11].Auto.Start )
      R_Coil( "MotorControl".Dev[11].Auto.CCWStart )
   END_RUNG
   RUNG wire#w3
      Contact( "MotorControl".Dev[12].Auto.Start )
      Contact( "AlwaysFALSE" )
      { S7_Templates := "time_type := Time" } "MotorData".Ton[1].TON(pt := "MotorData"."Time"[1], et =>)
      R_Coil( "MotorControl".Dev[12].Auto.Start )
      R_Coil( "MotorControl".Dev[12].Auto.CCWStart )
   END_RUNG
   RUNG wire#w2
      Contact( "AutoProcessControl".Global.H.EmptyPallet )
      R_Coil( "MotorControl".Dev[11].Auto.Start )
   END_RUNG
   RUNG wire#w1
      { S7_Templates := "SrcType := Time" } LT_Contact(in1 := "MotorData"."Time"[0], in2 := T#1M)
      Move(in := T#1M, out1 => "MotorData"."Time"[0])
   END_RUNG
   RUNG wire#w1
      { S7_Templates := "SrcType := Time" } LT_Contact(in1 := "MotorData"."Time"[1], in2 := T#1M)
      Move(in := T#1M, out1 => "MotorData"."Time"[1])
   END_RUNG
   // the same network as SCL:
   #_w1 := "AlwaysTRUE" AND "Station_Sys".Auto.Mode;
   #_w2 := #_w1 AND "PilzData"."85A2".I0 AND "PilzData"."85A2".I1;
   "MotorData".Ton[0].TON(IN := #_w2 AND "MotorControl".Dev[11].Auto.Start, PT := "MotorData"."Time"[0]);
   IF "MotorData".Ton[0].Q THEN
       "MotorControl".Dev[11].Auto.Start := FALSE;
       "MotorControl".Dev[11].Auto.CCWStart := FALSE;
   END_IF;
   "MotorData".Ton[1].TON(IN := #_w2 AND "MotorControl".Dev[12].Auto.Start AND "AlwaysFALSE",
                          PT := "MotorData"."Time"[1]);
   IF "MotorData".Ton[1].Q THEN
       "MotorControl".Dev[12].Auto.Start := FALSE;
       "MotorControl".Dev[12].Auto.CCWStart := FALSE;
   END_IF;
   IF #_w1 AND "AutoProcessControl".Global.H.EmptyPallet THEN
       "MotorControl".Dev[11].Auto.Start := FALSE;
   END_IF;
   IF "AlwaysTRUE" AND ("MotorData"."Time"[0] < T#1M) THEN "MotorData"."Time"[0] := T#1M; END_IF;
   IF "AlwaysTRUE" AND ("MotorData"."Time"[1] < T#1M) THEN "MotorData"."Time"[1] := T#1M; END_IF;
END_REGION

REGION Network 8: J-magnetLifting_Motor
   RUNG wire#powerrail
      "MotorContro_DB_2"(iAlwaysTrue := "AlwaysTRUE", iSysRun := "Station_Sys".Status.Run, iReset := "Station_Sys".Cmd.Reset, iAuto := "Station_Sys".Auto.Mode, iManual := "Station_Sys".Manual.Mode, i_ParySensor := 1, i_Alarm :=, iType := 1, i_RunInTimeDelay := T#20S, i_RunOutTimeDelay := T#20S, i_Interlock := 1, Control := "MotorControl".Dev[2])
   END_RUNG
   // the same network as SCL:
   "MotorContro_DB_2"(iAlwaysTrue := "AlwaysTRUE",   // "MotorContro"
                      iSysRun := "Station_Sys".Status.Run,
                      iReset := "Station_Sys".Cmd.Reset,
                      iAuto := "Station_Sys".Auto.Mode,
                      iManual := "Station_Sys".Manual.Mode,
                      i_ParySensor := 1,
                      iType := 1,
                      i_RunInTimeDelay := T#20S,
                      i_RunOutTimeDelay := T#20S,
                      i_Interlock := 1,
                      Control := "MotorControl".Dev[2]);
END_REGION

REGION Network 9 (SCL): J-magnetLifting_Motor_OutPut
   "oJ-magnetLifting_Start" := "MotorControl".Dev[2].OutControl.o_Start;
   "oJ-magnetLifting_CCWStart" := "MotorControl".Dev[2].OutControl.o_CCWStart;
   "oJ-magnetLifting_SpeedChange" := "MotorControl".Dev[2].OutControl.o_SpeedChanged;
END_REGION

REGION Network 10: J-MagnetLoad_Motor
   RUNG wire#powerrail
      "MotorContro_DB_13"(i_Interlock := wire#w1, iAlwaysTrue := "AlwaysTRUE", iSysRun := "Station_Sys".Status.Run, iReset := "Station_Sys".Cmd.Reset, iAuto := "Station_Sys".Auto.Mode, iManual := "Station_Sys".Manual.Mode, i_ParySensor := 1, i_Alarm :=, iType := 2, i_RunInTimeDelay := T#20S, i_RunOutTimeDelay := T#20S, Control := "MotorControl".Dev[13])
   END_RUNG
   RUNG wire#powerrail
      Contact( "PilzData"."85A2".I2 )
      Contact( "PilzData"."85A2".I3 )
      I_Contact( "PilzData"."85A3".I1 )
   END_RUNG wire#w1
   // the same network as SCL:
   "MotorContro_DB_13"(iAlwaysTrue := "AlwaysTRUE",   // "MotorContro"
                       iSysRun := "Station_Sys".Status.Run,
                       iReset := "Station_Sys".Cmd.Reset,
                       iAuto := "Station_Sys".Auto.Mode,
                       iManual := "Station_Sys".Manual.Mode,
                       i_ParySensor := 1,
                       iType := 2,
                       i_RunInTimeDelay := T#20S,
                       i_RunOutTimeDelay := T#20S,
                       i_Interlock := "PilzData"."85A2".I2 AND "PilzData"."85A2".I3 AND NOT "PilzData"."85A3".I1,
                       Control := "MotorControl".Dev[13]);
END_REGION

REGION Network 11: J-MagnetUnLoad_Motor
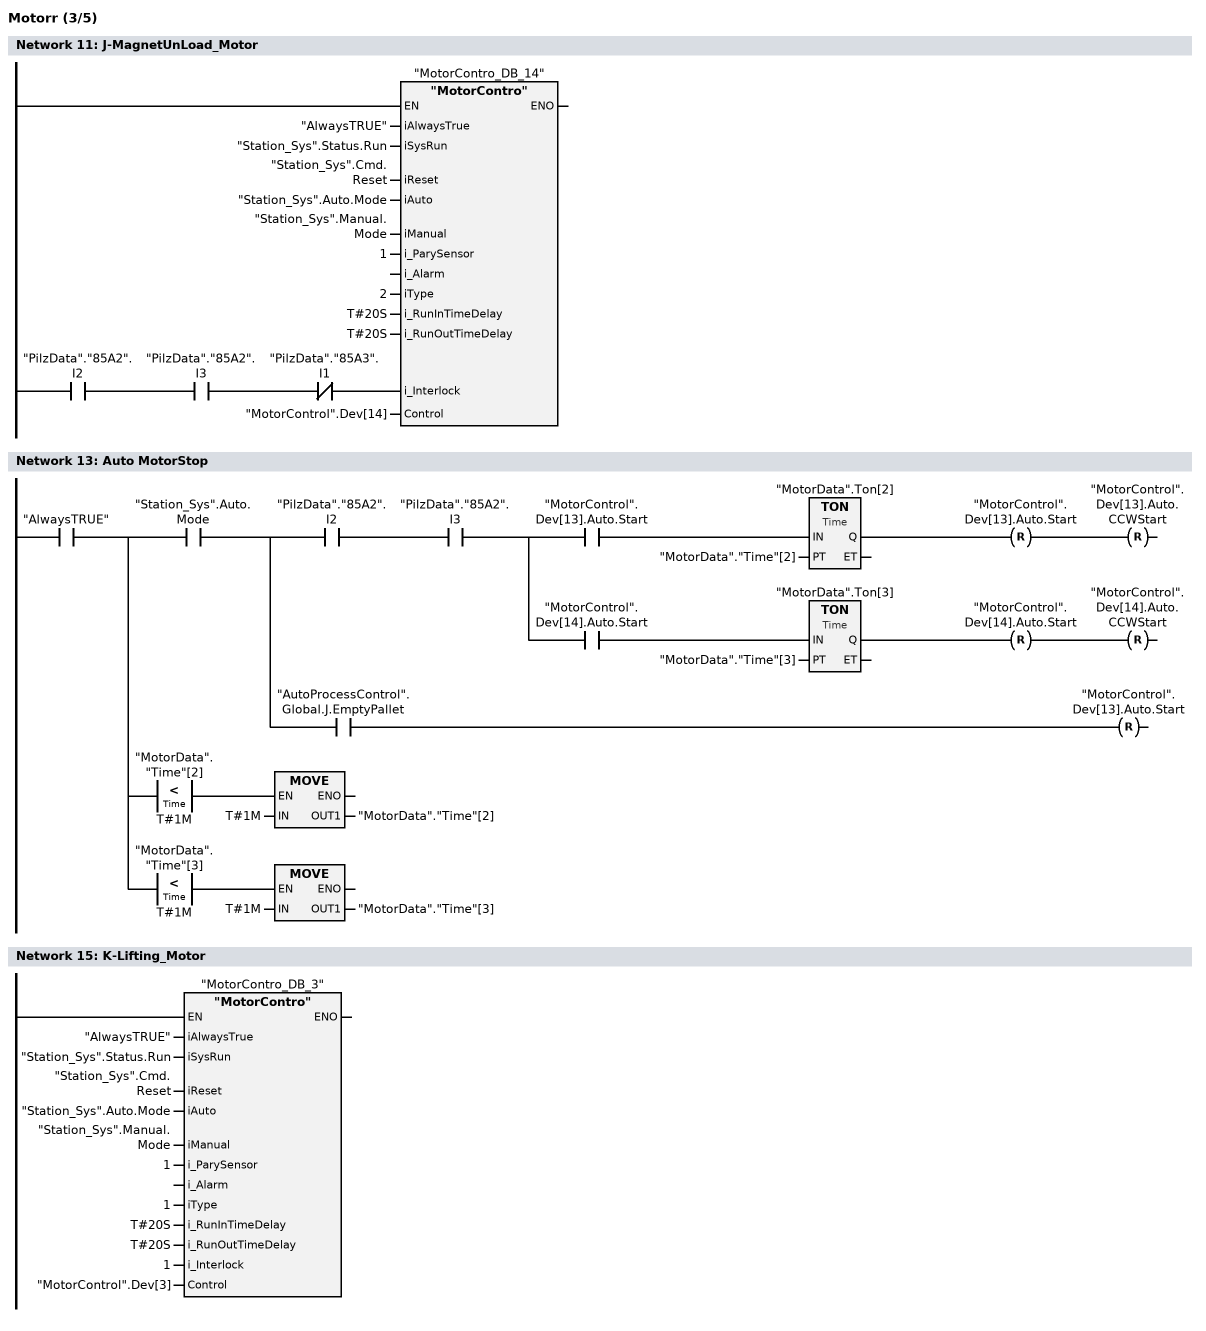
   RUNG wire#powerrail
      "MotorContro_DB_14"(i_Interlock := wire#w1, iAlwaysTrue := "AlwaysTRUE", iSysRun := "Station_Sys".Status.Run, iReset := "Station_Sys".Cmd.Reset, iAuto := "Station_Sys".Auto.Mode, iManual := "Station_Sys".Manual.Mode, i_ParySensor := 1, i_Alarm :=, iType := 2, i_RunInTimeDelay := T#20S, i_RunOutTimeDelay := T#20S, Control := "MotorControl".Dev[14])
   END_RUNG
   RUNG wire#powerrail
      Contact( "PilzData"."85A2".I2 )
      Contact( "PilzData"."85A2".I3 )
      I_Contact( "PilzData"."85A3".I1 )
   END_RUNG wire#w1
   // the same network as SCL:
   "MotorContro_DB_14"(iAlwaysTrue := "AlwaysTRUE",   // "MotorContro"
                       iSysRun := "Station_Sys".Status.Run,
                       iReset := "Station_Sys".Cmd.Reset,
                       iAuto := "Station_Sys".Auto.Mode,
                       iManual := "Station_Sys".Manual.Mode,
                       i_ParySensor := 1,
                       iType := 2,
                       i_RunInTimeDelay := T#20S,
                       i_RunOutTimeDelay := T#20S,
                       i_Interlock := "PilzData"."85A2".I2 AND "PilzData"."85A2".I3 AND NOT "PilzData"."85A3".I1,
                       Control := "MotorControl".Dev[14]);
END_REGION

REGION Network 12 (SCL): H-shaftLifting_Motor_OutPut / J-Magnet_Motor_OutPut
   "J-magnet Loading _CW" := "MotorControl".Dev[13].OutControl.o_Start;
   "J-magnet Loading _CCW" := "MotorControl".Dev[13].OutControl.o_CCWStart OR ("Station_Sys".Auto.Mode AND "AutoProcessControl".Global.J.EmptyPallet);

   "J-magnet Take _CW" := "MotorControl".Dev[14].OutControl.o_Start;
END_REGION

REGION Network 13: Auto MotorStop
   RUNG wire#powerrail
      Contact( "AlwaysTRUE" )
      wire#w1
      Contact( "Station_Sys".Auto.Mode )
      wire#w2
      Contact( "PilzData"."85A2".I2 )
      Contact( "PilzData"."85A2".I3 )
      wire#w3
      Contact( "MotorControl".Dev[13].Auto.Start )
      { S7_Templates := "time_type := Time" } "MotorData".Ton[2].TON(pt := "MotorData"."Time"[2], et =>)
      R_Coil( "MotorControl".Dev[13].Auto.Start )
      R_Coil( "MotorControl".Dev[13].Auto.CCWStart )
   END_RUNG
   RUNG wire#w3
      Contact( "MotorControl".Dev[14].Auto.Start )
      { S7_Templates := "time_type := Time" } "MotorData".Ton[3].TON(pt := "MotorData"."Time"[3], et =>)
      R_Coil( "MotorControl".Dev[14].Auto.Start )
      R_Coil( "MotorControl".Dev[14].Auto.CCWStart )
   END_RUNG
   RUNG wire#w2
      Contact( "AutoProcessControl".Global.J.EmptyPallet )
      R_Coil( "MotorControl".Dev[13].Auto.Start )
   END_RUNG
   RUNG wire#w1
      { S7_Templates := "SrcType := Time" } LT_Contact(in1 := "MotorData"."Time"[2], in2 := T#1M)
      Move(in := T#1M, out1 => "MotorData"."Time"[2])
   END_RUNG
   RUNG wire#w1
      { S7_Templates := "SrcType := Time" } LT_Contact(in1 := "MotorData"."Time"[3], in2 := T#1M)
      Move(in := T#1M, out1 => "MotorData"."Time"[3])
   END_RUNG
   // the same network as SCL:
   #_w1 := "AlwaysTRUE" AND "Station_Sys".Auto.Mode;
   #_w2 := #_w1 AND "PilzData"."85A2".I2 AND "PilzData"."85A2".I3;
   "MotorData".Ton[2].TON(IN := #_w2 AND "MotorControl".Dev[13].Auto.Start, PT := "MotorData"."Time"[2]);
   IF "MotorData".Ton[2].Q THEN
       "MotorControl".Dev[13].Auto.Start := FALSE;
       "MotorControl".Dev[13].Auto.CCWStart := FALSE;
   END_IF;
   "MotorData".Ton[3].TON(IN := #_w2 AND "MotorControl".Dev[14].Auto.Start, PT := "MotorData"."Time"[3]);
   IF "MotorData".Ton[3].Q THEN
       "MotorControl".Dev[14].Auto.Start := FALSE;
       "MotorControl".Dev[14].Auto.CCWStart := FALSE;
   END_IF;
   IF #_w1 AND "AutoProcessControl".Global.J.EmptyPallet THEN
       "MotorControl".Dev[13].Auto.Start := FALSE;
   END_IF;
   IF "AlwaysTRUE" AND ("MotorData"."Time"[2] < T#1M) THEN "MotorData"."Time"[2] := T#1M; END_IF;
   IF "AlwaysTRUE" AND ("MotorData"."Time"[3] < T#1M) THEN "MotorData"."Time"[3] := T#1M; END_IF;
END_REGION

REGION Network 15: K-Lifting_Motor
   RUNG wire#powerrail
      "MotorContro_DB_3"(iAlwaysTrue := "AlwaysTRUE", iSysRun := "Station_Sys".Status.Run, iReset := "Station_Sys".Cmd.Reset, iAuto := "Station_Sys".Auto.Mode, iManual := "Station_Sys".Manual.Mode, i_ParySensor := 1, i_Alarm :=, iType := 1, i_RunInTimeDelay := T#20S, i_RunOutTimeDelay := T#20S, i_Interlock := 1, Control := "MotorControl".Dev[3])
   END_RUNG
   // the same network as SCL:
   "MotorContro_DB_3"(iAlwaysTrue := "AlwaysTRUE",   // "MotorContro"
                      iSysRun := "Station_Sys".Status.Run,
                      iReset := "Station_Sys".Cmd.Reset,
                      iAuto := "Station_Sys".Auto.Mode,
                      iManual := "Station_Sys".Manual.Mode,
                      i_ParySensor := 1,
                      iType := 1,
                      i_RunInTimeDelay := T#20S,
                      i_RunOutTimeDelay := T#20S,
                      i_Interlock := 1,
                      Control := "MotorControl".Dev[3]);
END_REGION

REGION Network 16 (SCL): K-Lifting_Motor_OutPut
   "oK-Lifting3_Start" := "MotorControl".Dev[3].OutControl.o_Start;
   "oK-Lifting3_CCWStart" := "MotorControl".Dev[3].OutControl.o_CCWStart;
   "oK-Lifting3_SpeedChange" := "MotorControl".Dev[3].OutControl.o_SpeedChanged;
END_REGION

REGION Network 17: K-ReserveLoad_Motor
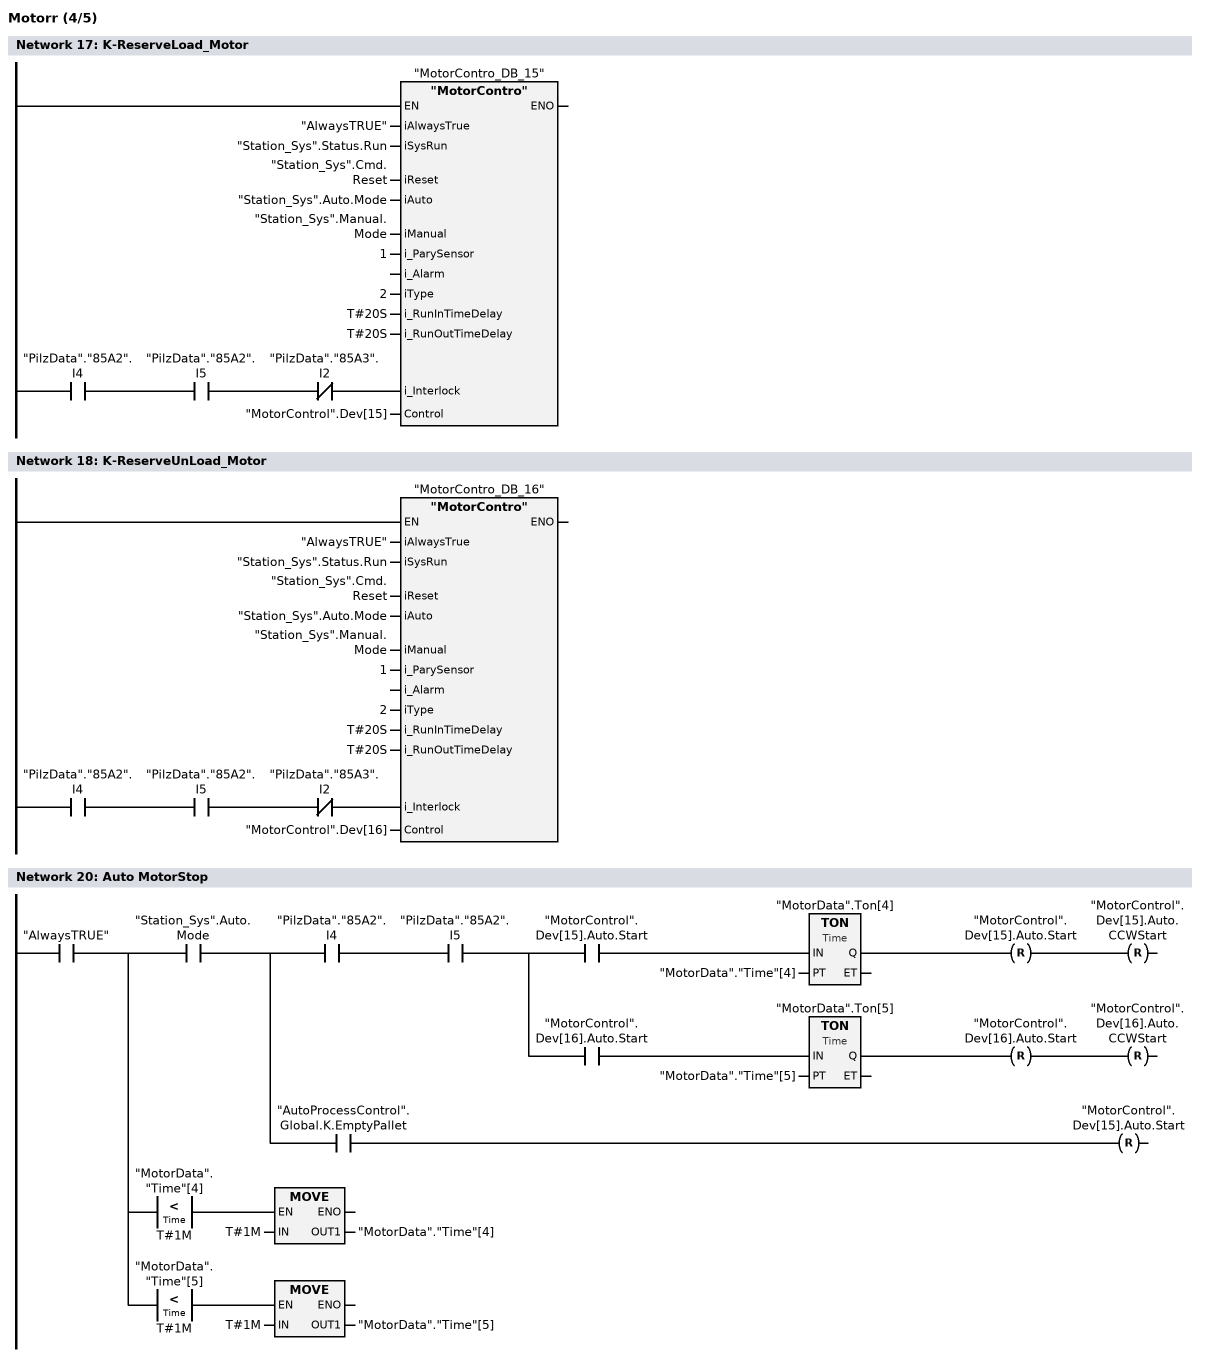
   RUNG wire#powerrail
      "MotorContro_DB_15"(i_Interlock := wire#w1, iAlwaysTrue := "AlwaysTRUE", iSysRun := "Station_Sys".Status.Run, iReset := "Station_Sys".Cmd.Reset, iAuto := "Station_Sys".Auto.Mode, iManual := "Station_Sys".Manual.Mode, i_ParySensor := 1, i_Alarm :=, iType := 2, i_RunInTimeDelay := T#20S, i_RunOutTimeDelay := T#20S, Control := "MotorControl".Dev[15])
   END_RUNG
   RUNG wire#powerrail
      Contact( "PilzData"."85A2".I4 )
      Contact( "PilzData"."85A2".I5 )
      I_Contact( "PilzData"."85A3".I2 )
   END_RUNG wire#w1
   // the same network as SCL:
   "MotorContro_DB_15"(iAlwaysTrue := "AlwaysTRUE",   // "MotorContro"
                       iSysRun := "Station_Sys".Status.Run,
                       iReset := "Station_Sys".Cmd.Reset,
                       iAuto := "Station_Sys".Auto.Mode,
                       iManual := "Station_Sys".Manual.Mode,
                       i_ParySensor := 1,
                       iType := 2,
                       i_RunInTimeDelay := T#20S,
                       i_RunOutTimeDelay := T#20S,
                       i_Interlock := "PilzData"."85A2".I4 AND "PilzData"."85A2".I5 AND NOT "PilzData"."85A3".I2,
                       Control := "MotorControl".Dev[15]);
END_REGION

REGION Network 18: K-ReserveUnLoad_Motor
   RUNG wire#powerrail
      "MotorContro_DB_16"(i_Interlock := wire#w1, iAlwaysTrue := "AlwaysTRUE", iSysRun := "Station_Sys".Status.Run, iReset := "Station_Sys".Cmd.Reset, iAuto := "Station_Sys".Auto.Mode, iManual := "Station_Sys".Manual.Mode, i_ParySensor := 1, i_Alarm :=, iType := 2, i_RunInTimeDelay := T#20S, i_RunOutTimeDelay := T#20S, Control := "MotorControl".Dev[16])
   END_RUNG
   RUNG wire#powerrail
      Contact( "PilzData"."85A2".I4 )
      Contact( "PilzData"."85A2".I5 )
      I_Contact( "PilzData"."85A3".I2 )
   END_RUNG wire#w1
   // the same network as SCL:
   "MotorContro_DB_16"(iAlwaysTrue := "AlwaysTRUE",   // "MotorContro"
                       iSysRun := "Station_Sys".Status.Run,
                       iReset := "Station_Sys".Cmd.Reset,
                       iAuto := "Station_Sys".Auto.Mode,
                       iManual := "Station_Sys".Manual.Mode,
                       i_ParySensor := 1,
                       iType := 2,
                       i_RunInTimeDelay := T#20S,
                       i_RunOutTimeDelay := T#20S,
                       i_Interlock := "PilzData"."85A2".I4 AND "PilzData"."85A2".I5 AND NOT "PilzData"."85A3".I2,
                       Control := "MotorControl".Dev[16]);
END_REGION

REGION Network 19 (SCL): H-shaftLifting_Motor_OutPut / K-Reserve_Motor_OutPut
   "K-Loading _CW" := "MotorControl".Dev[15].OutControl.o_Start;
   "K-Loading _CCW" := "MotorControl".Dev[15].OutControl.o_CCWStart OR ("Station_Sys".Auto.Mode AND "AutoProcessControl".Global.K.EmptyPallet);

   "K-Take _CW" := "MotorControl".Dev[16].OutControl.o_Start;
END_REGION

REGION Network 20: Auto MotorStop
   RUNG wire#powerrail
      Contact( "AlwaysTRUE" )
      wire#w1
      Contact( "Station_Sys".Auto.Mode )
      wire#w2
      Contact( "PilzData"."85A2".I4 )
      Contact( "PilzData"."85A2".I5 )
      wire#w3
      Contact( "MotorControl".Dev[15].Auto.Start )
      { S7_Templates := "time_type := Time" } "MotorData".Ton[4].TON(pt := "MotorData"."Time"[4], et =>)
      R_Coil( "MotorControl".Dev[15].Auto.Start )
      R_Coil( "MotorControl".Dev[15].Auto.CCWStart )
   END_RUNG
   RUNG wire#w3
      Contact( "MotorControl".Dev[16].Auto.Start )
      { S7_Templates := "time_type := Time" } "MotorData".Ton[5].TON(pt := "MotorData"."Time"[5], et =>)
      R_Coil( "MotorControl".Dev[16].Auto.Start )
      R_Coil( "MotorControl".Dev[16].Auto.CCWStart )
   END_RUNG
   RUNG wire#w2
      Contact( "AutoProcessControl".Global.K.EmptyPallet )
      R_Coil( "MotorControl".Dev[15].Auto.Start )
   END_RUNG
   RUNG wire#w1
      { S7_Templates := "SrcType := Time" } LT_Contact(in1 := "MotorData"."Time"[4], in2 := T#1M)
      Move(in := T#1M, out1 => "MotorData"."Time"[4])
   END_RUNG
   RUNG wire#w1
      { S7_Templates := "SrcType := Time" } LT_Contact(in1 := "MotorData"."Time"[5], in2 := T#1M)
      Move(in := T#1M, out1 => "MotorData"."Time"[5])
   END_RUNG
   // the same network as SCL:
   #_w1 := "AlwaysTRUE" AND "Station_Sys".Auto.Mode;
   #_w2 := #_w1 AND "PilzData"."85A2".I4 AND "PilzData"."85A2".I5;
   "MotorData".Ton[4].TON(IN := #_w2 AND "MotorControl".Dev[15].Auto.Start, PT := "MotorData"."Time"[4]);
   IF "MotorData".Ton[4].Q THEN
       "MotorControl".Dev[15].Auto.Start := FALSE;
       "MotorControl".Dev[15].Auto.CCWStart := FALSE;
   END_IF;
   "MotorData".Ton[5].TON(IN := #_w2 AND "MotorControl".Dev[16].Auto.Start, PT := "MotorData"."Time"[5]);
   IF "MotorData".Ton[5].Q THEN
       "MotorControl".Dev[16].Auto.Start := FALSE;
       "MotorControl".Dev[16].Auto.CCWStart := FALSE;
   END_IF;
   IF #_w1 AND "AutoProcessControl".Global.K.EmptyPallet THEN
       "MotorControl".Dev[15].Auto.Start := FALSE;
   END_IF;
   IF "AlwaysTRUE" AND ("MotorData"."Time"[4] < T#1M) THEN "MotorData"."Time"[4] := T#1M; END_IF;
   IF "AlwaysTRUE" AND ("MotorData"."Time"[5] < T#1M) THEN "MotorData"."Time"[5] := T#1M; END_IF;
END_REGION

REGION Network 22: L-Unloading_Motor
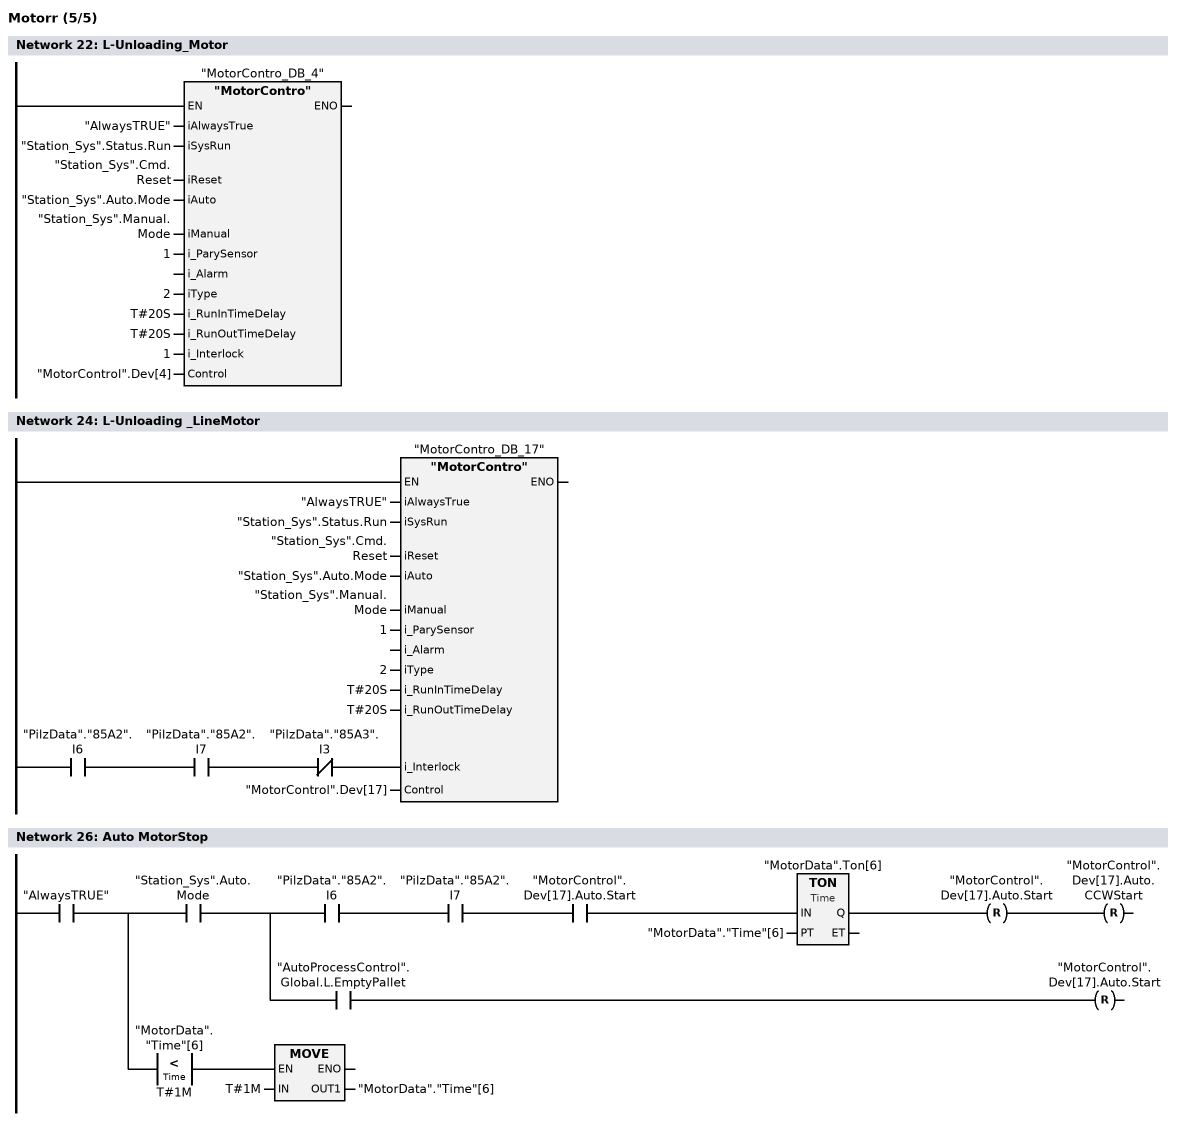
   RUNG wire#powerrail
      "MotorContro_DB_4"(iAlwaysTrue := "AlwaysTRUE", iSysRun := "Station_Sys".Status.Run, iReset := "Station_Sys".Cmd.Reset, iAuto := "Station_Sys".Auto.Mode, iManual := "Station_Sys".Manual.Mode, i_ParySensor := 1, i_Alarm :=, iType := 2, i_RunInTimeDelay := T#20S, i_RunOutTimeDelay := T#20S, i_Interlock := 1, Control := "MotorControl".Dev[4])
   END_RUNG
   // the same network as SCL:
   "MotorContro_DB_4"(iAlwaysTrue := "AlwaysTRUE",   // "MotorContro"
                      iSysRun := "Station_Sys".Status.Run,
                      iReset := "Station_Sys".Cmd.Reset,
                      iAuto := "Station_Sys".Auto.Mode,
                      iManual := "Station_Sys".Manual.Mode,
                      i_ParySensor := 1,
                      iType := 2,
                      i_RunInTimeDelay := T#20S,
                      i_RunOutTimeDelay := T#20S,
                      i_Interlock := 1,
                      Control := "MotorControl".Dev[4]);
END_REGION

REGION Network 23 (SCL): L-Unloading_Motor_OutPut
   "oL-Unloading_CW" := "MotorControl".Dev[4].OutControl.o_Start;
   "oL-Unloading_CCW" := "MotorControl".Dev[4].OutControl.o_CCWStart;
END_REGION

REGION Network 24: L-Unloading _LineMotor
   RUNG wire#powerrail
      "MotorContro_DB_17"(i_Interlock := wire#w1, iAlwaysTrue := "AlwaysTRUE", iSysRun := "Station_Sys".Status.Run, iReset := "Station_Sys".Cmd.Reset, iAuto := "Station_Sys".Auto.Mode, iManual := "Station_Sys".Manual.Mode, i_ParySensor := 1, i_Alarm :=, iType := 2, i_RunInTimeDelay := T#20S, i_RunOutTimeDelay := T#20S, Control := "MotorControl".Dev[17])
   END_RUNG
   RUNG wire#powerrail
      Contact( "PilzData"."85A2".I6 )
      Contact( "PilzData"."85A2".I7 )
      I_Contact( "PilzData"."85A3".I3 )
   END_RUNG wire#w1
   // the same network as SCL:
   "MotorContro_DB_17"(iAlwaysTrue := "AlwaysTRUE",   // "MotorContro"
                       iSysRun := "Station_Sys".Status.Run,
                       iReset := "Station_Sys".Cmd.Reset,
                       iAuto := "Station_Sys".Auto.Mode,
                       iManual := "Station_Sys".Manual.Mode,
                       i_ParySensor := 1,
                       iType := 2,
                       i_RunInTimeDelay := T#20S,
                       i_RunOutTimeDelay := T#20S,
                       i_Interlock := "PilzData"."85A2".I6 AND "PilzData"."85A2".I7 AND NOT "PilzData"."85A3".I3,
                       Control := "MotorControl".Dev[17]);
END_REGION

REGION Network 25 (SCL): H-shaftLifting_Motor_OutPut / L-Unloading _LineMotor_OutPut
   "L-Unloading _LineMotor_CW" := "MotorControl".Dev[17].OutControl.o_Start;
   "L-Unloading _LineMotor_CCW" := "MotorControl".Dev[17].OutControl.o_CCWStart OR ("Station_Sys".Auto.Mode AND "AutoProcessControl".Global.L.EmptyPallet);
END_REGION

REGION Network 26: Auto MotorStop
   RUNG wire#powerrail
      Contact( "AlwaysTRUE" )
      wire#w1
      Contact( "Station_Sys".Auto.Mode )
      wire#w2
      Contact( "PilzData"."85A2".I6 )
      Contact( "PilzData"."85A2".I7 )
      Contact( "MotorControl".Dev[17].Auto.Start )
      { S7_Templates := "time_type := Time" } "MotorData".Ton[6].TON(pt := "MotorData"."Time"[6], et =>)
      R_Coil( "MotorControl".Dev[17].Auto.Start )
      R_Coil( "MotorControl".Dev[17].Auto.CCWStart )
   END_RUNG
   RUNG wire#w2
      Contact( "AutoProcessControl".Global.L.EmptyPallet )
      R_Coil( "MotorControl".Dev[17].Auto.Start )
   END_RUNG
   RUNG wire#w1
      { S7_Templates := "SrcType := Time" } LT_Contact(in1 := "MotorData"."Time"[6], in2 := T#1M)
      Move(in := T#1M, out1 => "MotorData"."Time"[6])
   END_RUNG
   // the same network as SCL:
   #_w1 := "AlwaysTRUE" AND "Station_Sys".Auto.Mode;
   "MotorData".Ton[6].TON(IN := #_w1 AND "PilzData"."85A2".I6 AND "PilzData"."85A2".I7 AND "MotorControl".Dev[17].Auto.Start,
                          PT := "MotorData"."Time"[6]);
   IF "MotorData".Ton[6].Q THEN
       "MotorControl".Dev[17].Auto.Start := FALSE;
       "MotorControl".Dev[17].Auto.CCWStart := FALSE;
   END_IF;
   IF #_w1 AND "AutoProcessControl".Global.L.EmptyPallet THEN
       "MotorControl".Dev[17].Auto.Start := FALSE;
   END_IF;
   IF "AlwaysTRUE" AND ("MotorData"."Time"[6] < T#1M) THEN "MotorData"."Time"[6] := T#1M; END_IF;
END_REGION
END_FUNCTION

FUNCTION_BLOCK "MotorContro"   // FB3100, LAD
{ S7_Optimized_Access := 'TRUE' }
// stored: AutoNumber false, MemoryReserve 100, SetENOAutomatically false
   VAR_INPUT
      iAlwaysTrue : Bool;
      iSysRun : Bool;
      iReset : Bool;
      iAuto : Bool;
      iManual : Bool;
      i_ParySensor : Bool;
      i_Alarm : Bool;
      iType : Int;
      i_RunInTimeDelay : Time;
      i_RunOutTimeDelay : Time;
      i_Interlock : Bool;
   END_VAR
   VAR_IN_OUT
      Control : "Motor_Control";
   END_VAR
   VAR
      TON : Array[0..5] of TON_TIME;
      Zero { S7_SetPoint := 'True'} : Array[0..15] of Bool;
   END_VAR
   VAR_TEMP   // added for the SCL form of the ladder/FBD networks
      _w1 : Bool;
   END_VAR
BEGIN

REGION Network 1: Reset
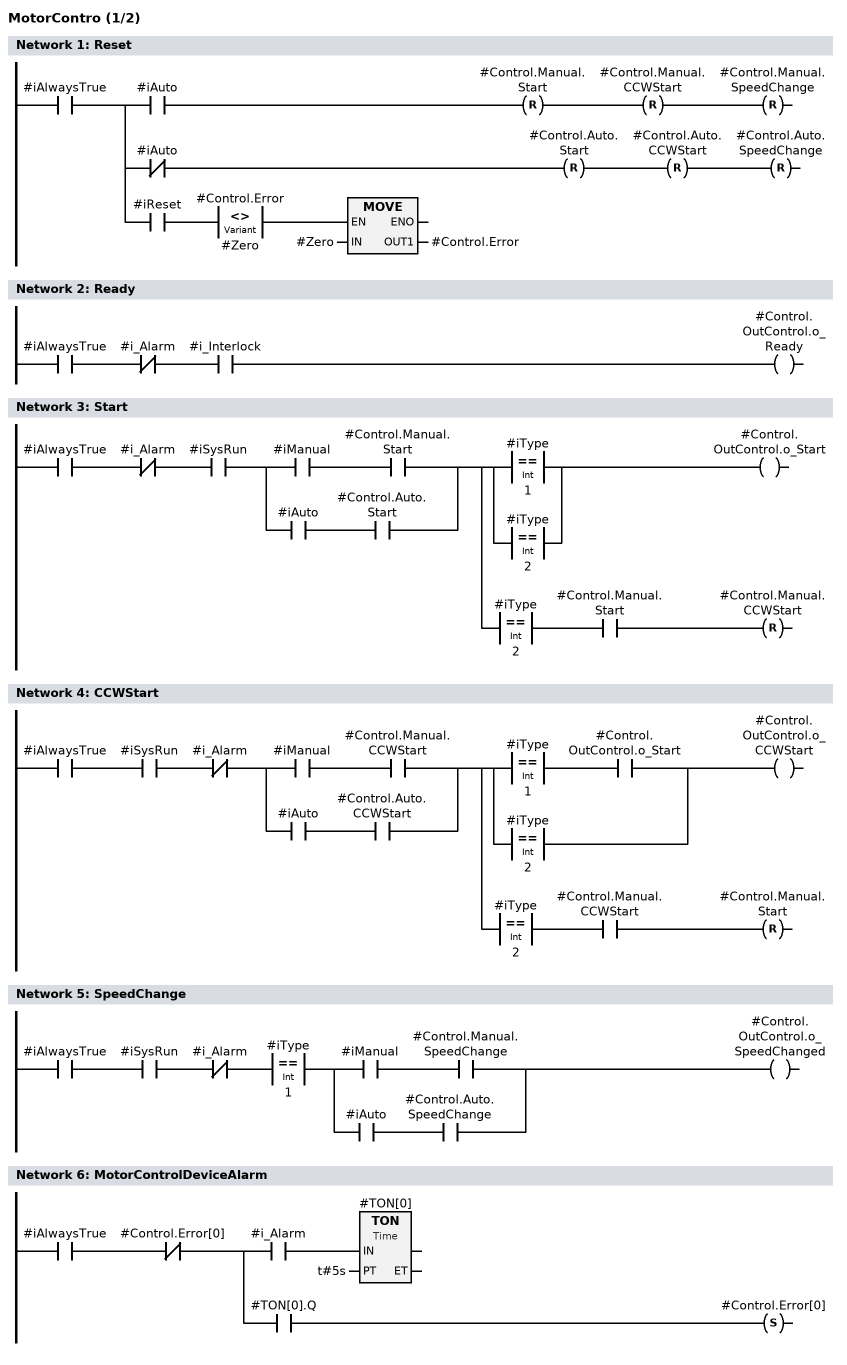
   RUNG wire#powerrail
      Contact( #iAlwaysTrue )
      wire#w1
      Contact( #iAuto )
      R_Coil( #Control.Manual.Start )
      R_Coil( #Control.Manual.CCWStart )
      R_Coil( #Control.Manual.SpeedChange )
   END_RUNG
   RUNG wire#w1
      I_Contact( #iAuto )
      R_Coil( #Control.Auto.Start )
      R_Coil( #Control.Auto.CCWStart )
      R_Coil( #Control.Auto.SpeedChange )
   END_RUNG
   RUNG wire#w1
      Contact( #iReset )
      { S7_Templates := "SrcType := Variant" } NE_Contact(in1 := #Control.Error, in2 := #Zero)
      Move(in := #Zero, out1 => #Control.Error)
   END_RUNG
   // the same network as SCL:
   IF #iAlwaysTrue AND #iAuto THEN
       #Control.Manual.Start := FALSE;
       #Control.Manual.CCWStart := FALSE;
       #Control.Manual.SpeedChange := FALSE;
   END_IF;
   IF #iAlwaysTrue AND NOT #iAuto THEN
       #Control.Auto.Start := FALSE;
       #Control.Auto.CCWStart := FALSE;
       #Control.Auto.SpeedChange := FALSE;
   END_IF;
   IF #iAlwaysTrue AND #iReset AND (#Control.Error <> #Zero) THEN #Control.Error := #Zero; END_IF;
END_REGION

REGION Network 2: Ready
   RUNG wire#powerrail
      Contact( #iAlwaysTrue )
      I_Contact( #i_Alarm )
      Contact( #i_Interlock )
      Coil( #Control.OutControl.o_Ready )
   END_RUNG
   // the same network as SCL:
   #Control.OutControl.o_Ready := #iAlwaysTrue AND NOT #i_Alarm AND #i_Interlock;
END_REGION

REGION Network 3: Start
   RUNG wire#powerrail
      Contact( #iAlwaysTrue )
      I_Contact( #i_Alarm )
      Contact( #iSysRun )
      wire#w1
      Contact( #iManual )
      Contact( #Control.Manual.Start )
      wire#w2
      { S7_Templates := "SrcType := Int" } EQ_Contact(in1 := #iType, in2 := 1)
      wire#w3
      Coil( #Control.OutControl.o_Start )
   END_RUNG
   RUNG wire#w1
      Contact( #iAuto )
      Contact( #Control.Auto.Start )
   END_RUNG wire#w2
   RUNG wire#w2
      { S7_Templates := "SrcType := Int" } EQ_Contact(in1 := #iType, in2 := 2)
   END_RUNG wire#w3
   RUNG wire#w2
      { S7_Templates := "SrcType := Int" } EQ_Contact(in1 := #iType, in2 := 2)
      Contact( #Control.Manual.Start )
      R_Coil( #Control.Manual.CCWStart )
   END_RUNG
   // the same network as SCL:
   #_w1 := #iAlwaysTrue AND NOT #i_Alarm AND #iSysRun AND ((#iManual AND #Control.Manual.Start) OR (#iAuto AND #Control.Auto.Start));
   #Control.OutControl.o_Start := #_w1 AND ((#iType = 1) OR (#iType = 2));
   IF #_w1 AND (#iType = 2) AND #Control.Manual.Start THEN #Control.Manual.CCWStart := FALSE; END_IF;
END_REGION

REGION Network 4: CCWStart
   RUNG wire#powerrail
      Contact( #iAlwaysTrue )
      Contact( #iSysRun )
      I_Contact( #i_Alarm )
      wire#w1
      Contact( #iManual )
      Contact( #Control.Manual.CCWStart )
      wire#w2
      { S7_Templates := "SrcType := Int" } EQ_Contact(in1 := #iType, in2 := 1)
      Contact( #Control.OutControl.o_Start )
      wire#w3
      Coil( #Control.OutControl.o_CCWStart )
   END_RUNG
   RUNG wire#w1
      Contact( #iAuto )
      Contact( #Control.Auto.CCWStart )
   END_RUNG wire#w2
   RUNG wire#w2
      { S7_Templates := "SrcType := Int" } EQ_Contact(in1 := #iType, in2 := 2)
   END_RUNG wire#w3
   RUNG wire#w2
      { S7_Templates := "SrcType := Int" } EQ_Contact(in1 := #iType, in2 := 2)
      Contact( #Control.Manual.CCWStart )
      R_Coil( #Control.Manual.Start )
   END_RUNG
   // the same network as SCL:
   #_w1 := #iAlwaysTrue AND #iSysRun AND NOT #i_Alarm AND ((#iManual AND #Control.Manual.CCWStart) OR (#iAuto AND #Control.Auto.CCWStart));
   #Control.OutControl.o_CCWStart := #_w1 AND (((#iType = 1) AND #Control.OutControl.o_Start) OR (#iType = 2));
   IF #_w1 AND (#iType = 2) AND #Control.Manual.CCWStart THEN #Control.Manual.Start := FALSE; END_IF;
END_REGION

REGION Network 5: SpeedChange
   RUNG wire#powerrail
      Contact( #iAlwaysTrue )
      Contact( #iSysRun )
      I_Contact( #i_Alarm )
      { S7_Templates := "SrcType := Int" } EQ_Contact(in1 := #iType, in2 := 1)
      wire#w1
      Contact( #iManual )
      Contact( #Control.Manual.SpeedChange )
      wire#w2
      Coil( #Control.OutControl.o_SpeedChanged )
   END_RUNG
   RUNG wire#w1
      Contact( #iAuto )
      Contact( #Control.Auto.SpeedChange )
   END_RUNG wire#w2
   // the same network as SCL:
   #Control.OutControl.o_SpeedChanged := #iAlwaysTrue AND #iSysRun AND NOT #i_Alarm AND (#iType = 1) AND ((#iManual AND #Control.Manual.SpeedChange) OR (#iAuto AND #Control.Auto.SpeedChange));
END_REGION

REGION Network 6: MotorControlDeviceAlarm
   RUNG wire#powerrail
      Contact( #iAlwaysTrue )
      I_Contact( #Control.Error[0] )
      wire#w1
      Contact( #i_Alarm )
      { S7_Templates := "time_type := Time" } #TON[0].TON(pt := t#5s, et =>)
   END_RUNG
   RUNG wire#w1
      Contact( #TON[0].Q )
      S_Coil( #Control.Error[0] )
   END_RUNG
   // the same network as SCL:
   #_w1 := #iAlwaysTrue AND NOT #Control.Error[0];
   #TON[0].TON(IN := #_w1 AND #i_Alarm, PT := t#5s);
   IF #_w1 AND #TON[0].Q THEN #Control.Error[0] := TRUE; END_IF;
END_REGION

REGION Network 7: PalletRunInTimeOut
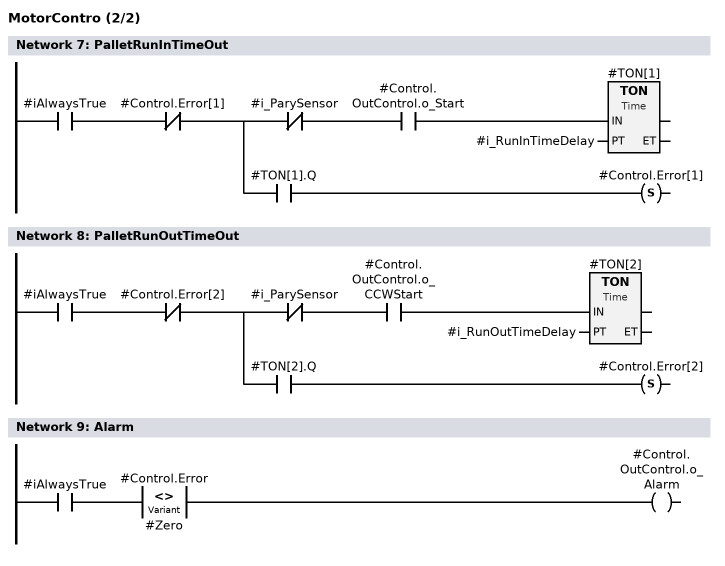
   RUNG wire#powerrail
      Contact( #iAlwaysTrue )
      I_Contact( #Control.Error[1] )
      wire#w1
      I_Contact( #i_ParySensor )
      Contact( #Control.OutControl.o_Start )
      { S7_Templates := "time_type := Time" } #TON[1].TON(pt := #i_RunInTimeDelay, et =>)
   END_RUNG
   RUNG wire#w1
      Contact( #TON[1].Q )
      S_Coil( #Control.Error[1] )
   END_RUNG
   // the same network as SCL:
   #_w1 := #iAlwaysTrue AND NOT #Control.Error[1];
   #TON[1].TON(IN := #_w1 AND NOT #i_ParySensor AND #Control.OutControl.o_Start, PT := #i_RunInTimeDelay);
   IF #_w1 AND #TON[1].Q THEN #Control.Error[1] := TRUE; END_IF;
END_REGION

REGION Network 8: PalletRunOutTimeOut
   RUNG wire#powerrail
      Contact( #iAlwaysTrue )
      I_Contact( #Control.Error[2] )
      wire#w1
      I_Contact( #i_ParySensor )
      Contact( #Control.OutControl.o_CCWStart )
      { S7_Templates := "time_type := Time" } #TON[2].TON(pt := #i_RunOutTimeDelay, et =>)
   END_RUNG
   RUNG wire#w1
      Contact( #TON[2].Q )
      S_Coil( #Control.Error[2] )
   END_RUNG
   // the same network as SCL:
   #_w1 := #iAlwaysTrue AND NOT #Control.Error[2];
   #TON[2].TON(IN := #_w1 AND NOT #i_ParySensor AND #Control.OutControl.o_CCWStart, PT := #i_RunOutTimeDelay);
   IF #_w1 AND #TON[2].Q THEN #Control.Error[2] := TRUE; END_IF;
END_REGION

REGION Network 9: Alarm
   RUNG wire#powerrail
      Contact( #iAlwaysTrue )
      { S7_Templates := "SrcType := Variant" } NE_Contact(in1 := #Control.Error, in2 := #Zero)
      Coil( #Control.OutControl.o_Alarm )
   END_RUNG
   // the same network as SCL:
   #Control.OutControl.o_Alarm := #iAlwaysTrue AND (#Control.Error <> #Zero);
END_REGION
END_FUNCTION_BLOCK

FUNCTION "Stopper" : Void   // FC2600, LAD
{ S7_Optimized_Access := 'TRUE' }
// stored: AutoNumber false, SetENOAutomatically false
BEGIN
END_FUNCTION

FUNCTION "Pilz" : Void   // FC2700, LAD
{ S7_Optimized_Access := 'TRUE' }
VERSION : 0.1
// stored: AutoNumber false, IsIECCheckEnabled false, SetENOAutomatically false, UDAEnableTagReadback false
   VAR_TEMP
      Ret_Val_1 : Int;
      Ret_Val_2 : Int;
      Ret_Val_3 : Int;
      Ret_Val_4 : Int;
   END_VAR
   VAR_TEMP   // added for the SCL form of the ladder/FBD networks
      _w1 : Bool;
   END_VAR
BEGIN

REGION Network 1: 功能块调用 / Pilz
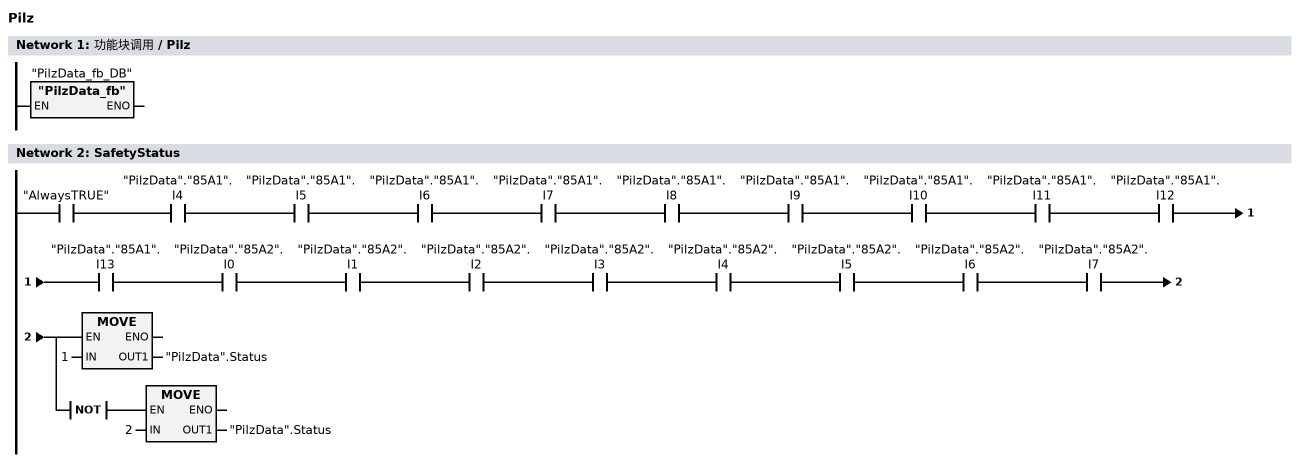
   RUNG wire#powerrail
      "PilzData_fb_DB"()
   END_RUNG
   // the same network as SCL:
   "PilzData_fb_DB"();   // "PilzData_fb"
END_REGION

REGION Network 2: SafetyStatus
   RUNG wire#powerrail
      Contact( "AlwaysTRUE" )
      Contact( "PilzData"."85A1".I4 )
      Contact( "PilzData"."85A1".I5 )
      Contact( "PilzData"."85A1".I6 )
      Contact( "PilzData"."85A1".I7 )
      Contact( "PilzData"."85A1".I8 )
      Contact( "PilzData"."85A1".I9 )
      Contact( "PilzData"."85A1".I10 )
      Contact( "PilzData"."85A1".I11 )
      Contact( "PilzData"."85A1".I12 )
      Contact( "PilzData"."85A1".I13 )
      Contact( "PilzData"."85A2".I0 )
      Contact( "PilzData"."85A2".I1 )
      Contact( "PilzData"."85A2".I2 )
      Contact( "PilzData"."85A2".I3 )
      Contact( "PilzData"."85A2".I4 )
      Contact( "PilzData"."85A2".I5 )
      Contact( "PilzData"."85A2".I6 )
      Contact( "PilzData"."85A2".I7 )
      wire#w1
      Move(in := 1, out1 => "PilzData".Status)
   END_RUNG
   RUNG wire#w1
      Not()
      Move(in := 2, out1 => "PilzData".Status)
   END_RUNG
   // the same network as SCL:
   #_w1 := "AlwaysTRUE" AND "PilzData"."85A1".I4 AND "PilzData"."85A1".I5 AND "PilzData"."85A1".I6 AND "PilzData"."85A1".I7 AND "PilzData"."85A1".I8 AND "PilzData"."85A1".I9 AND "PilzData"."85A1".I10 AND "PilzData"."85A1".I11 AND "PilzData"."85A1".I12 AND "PilzData"."85A1".I13 AND "PilzData"."85A2".I0 AND "PilzData"."85A2".I1 AND "PilzData"."85A2".I2 AND "PilzData"."85A2".I3 AND "PilzData"."85A2".I4 AND "PilzData"."85A2".I5 AND "PilzData"."85A2".I6 AND "PilzData"."85A2".I7;
   IF #_w1 THEN "PilzData".Status := 1; END_IF;
   IF NOT #_w1 THEN "PilzData".Status := 2; END_IF;
END_REGION
END_FUNCTION

FUNCTION "Gluing" : Void   // FC2800, LAD
{ S7_Optimized_Access := 'TRUE' }
// stored: AutoNumber false, SetENOAutomatically false
   VAR_TEMP   // added for the SCL form of the ladder/FBD networks
      _w1 : Bool;
      _w2 : Bool;
   END_VAR
BEGIN

REGION Network 1 (SCL): Input and Output
   //   Input
   "GluingControl".Input.GluingDeviceReady := "iC- GluingDeviceReady";
   "GluingControl".Input.GluingFault := "iC- GluingFault";
   "GluingControl".Input.GluingRefillTank := "iC- GluingRefillTank";
   "GluingControl".Input.GluingTankEmpty := "iC- GluingTankEmpty";

   //   Output
   "oC-GluingPro_X" := "GluingControl".Output.GluingPro_X;
   "oC-GluingPro_Y" := "GluingControl".Output.GluingPro_Y;
   "oC-GluingPro_Z" := "GluingControl".Output.GluingPro_Z;
   "oC-GluingReset" := "GluingControl".Output.GluingReset;
END_REGION

REGION Network 2: Reset
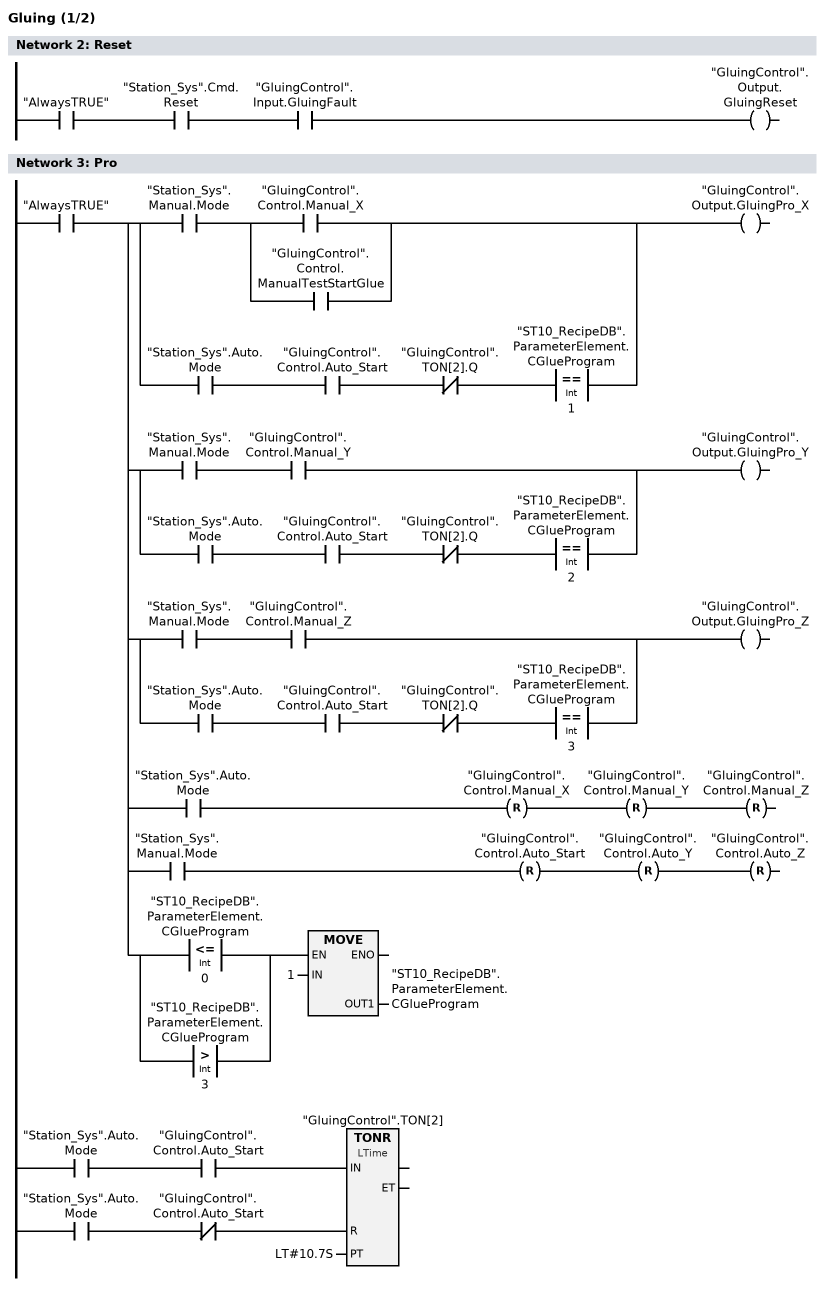
   RUNG wire#powerrail
      Contact( "AlwaysTRUE" )
      Contact( "Station_Sys".Cmd.Reset )
      Contact( "GluingControl".Input.GluingFault )
      Coil( "GluingControl".Output.GluingReset )
   END_RUNG
   // the same network as SCL:
   "GluingControl".Output.GluingReset := "AlwaysTRUE" AND "Station_Sys".Cmd.Reset AND "GluingControl".Input.GluingFault;
END_REGION

REGION Network 3: Pro
   RUNG wire#powerrail
      Contact( "AlwaysTRUE" )
      wire#w1
      Contact( "Station_Sys".Manual.Mode )
      wire#w2
      Contact( "GluingControl".Control.Manual_X )
      wire#w3
      Coil( "GluingControl".Output.GluingPro_X )
   END_RUNG
   RUNG wire#w2
      Contact( "GluingControl".Control.ManualTestStartGlue )
   END_RUNG wire#w3
   RUNG wire#w1
      Contact( "Station_Sys".Auto.Mode )
      Contact( "GluingControl".Control.Auto_Start )
      I_Contact( "GluingControl".TON[2].Q )
      { S7_Templates := "SrcType := Int" } EQ_Contact(in1 := "ST10_RecipeDB".ParameterElement.CGlueProgram, in2 := 1)
   END_RUNG wire#w3
   RUNG wire#w1
      Contact( "Station_Sys".Manual.Mode )
      Contact( "GluingControl".Control.Manual_Y )
      wire#w4
      Coil( "GluingControl".Output.GluingPro_Y )
   END_RUNG
   RUNG wire#w1
      Contact( "Station_Sys".Auto.Mode )
      Contact( "GluingControl".Control.Auto_Start )
      I_Contact( "GluingControl".TON[2].Q )
      { S7_Templates := "SrcType := Int" } EQ_Contact(in1 := "ST10_RecipeDB".ParameterElement.CGlueProgram, in2 := 2)
   END_RUNG wire#w4
   RUNG wire#w1
      Contact( "Station_Sys".Manual.Mode )
      Contact( "GluingControl".Control.Manual_Z )
      wire#w5
      Coil( "GluingControl".Output.GluingPro_Z )
   END_RUNG
   RUNG wire#w1
      Contact( "Station_Sys".Auto.Mode )
      Contact( "GluingControl".Control.Auto_Start )
      I_Contact( "GluingControl".TON[2].Q )
      { S7_Templates := "SrcType := Int" } EQ_Contact(in1 := "ST10_RecipeDB".ParameterElement.CGlueProgram, in2 := 3)
   END_RUNG wire#w5
   RUNG wire#w1
      Contact( "Station_Sys".Auto.Mode )
      R_Coil( "GluingControl".Control.Manual_X )
      R_Coil( "GluingControl".Control.Manual_Y )
      R_Coil( "GluingControl".Control.Manual_Z )
   END_RUNG
   RUNG wire#w1
      Contact( "Station_Sys".Manual.Mode )
      R_Coil( "GluingControl".Control.Auto_Start )
      R_Coil( "GluingControl".Control.Auto_Y )
      R_Coil( "GluingControl".Control.Auto_Z )
   END_RUNG
   RUNG wire#w1
      { S7_Templates := "SrcType := Int" } LE_Contact(in1 := "ST10_RecipeDB".ParameterElement.CGlueProgram, in2 := 0)
      wire#w6
      Move(in := 1, out1 => "ST10_RecipeDB".ParameterElement.CGlueProgram)
   END_RUNG
   RUNG wire#w1
      { S7_Templates := "SrcType := Int" } GT_Contact(in1 := "ST10_RecipeDB".ParameterElement.CGlueProgram, in2 := 3)
   END_RUNG wire#w6
   RUNG wire#powerrail
      Contact( "Station_Sys".Auto.Mode )
      Contact( "GluingControl".Control.Auto_Start )
      { S7_Templates := "time_type := LTime" } "GluingControl".TON[2].TONR(r := wire#w7, pt := LT#10.7S, et =>)
   END_RUNG
   RUNG wire#powerrail
      Contact( "Station_Sys".Auto.Mode )
      I_Contact( "GluingControl".Control.Auto_Start )
   END_RUNG wire#w7
   // the same network as SCL:
   "GluingControl".Output.GluingPro_X := "AlwaysTRUE" AND (("Station_Sys".Manual.Mode AND ("GluingControl".Control.Manual_X OR "GluingControl".Control.ManualTestStartGlue)) OR ("Station_Sys".Auto.Mode AND "GluingControl".Control.Auto_Start AND NOT "GluingControl".TON[2].Q AND ("ST10_RecipeDB".ParameterElement.CGlueProgram = 1)));
   "GluingControl".Output.GluingPro_Y := "AlwaysTRUE" AND (("Station_Sys".Manual.Mode AND "GluingControl".Control.Manual_Y) OR ("Station_Sys".Auto.Mode AND "GluingControl".Control.Auto_Start AND NOT "GluingControl".TON[2].Q AND ("ST10_RecipeDB".ParameterElement.CGlueProgram = 2)));
   "GluingControl".Output.GluingPro_Z := "AlwaysTRUE" AND (("Station_Sys".Manual.Mode AND "GluingControl".Control.Manual_Z) OR ("Station_Sys".Auto.Mode AND "GluingControl".Control.Auto_Start AND NOT "GluingControl".TON[2].Q AND ("ST10_RecipeDB".ParameterElement.CGlueProgram = 3)));
   IF "AlwaysTRUE" AND "Station_Sys".Auto.Mode THEN
       "GluingControl".Control.Manual_X := FALSE;
       "GluingControl".Control.Manual_Y := FALSE;
       "GluingControl".Control.Manual_Z := FALSE;
   END_IF;
   IF "AlwaysTRUE" AND "Station_Sys".Manual.Mode THEN
       "GluingControl".Control.Auto_Start := FALSE;
       "GluingControl".Control.Auto_Y := FALSE;
       "GluingControl".Control.Auto_Z := FALSE;
   END_IF;
   IF "AlwaysTRUE" AND (("ST10_RecipeDB".ParameterElement.CGlueProgram <= 0) OR ("ST10_RecipeDB".ParameterElement.CGlueProgram > 3)) THEN
       "ST10_RecipeDB".ParameterElement.CGlueProgram := 1;
   END_IF;
   "GluingControl".TON[2].TONR(IN := "Station_Sys".Auto.Mode AND "GluingControl".Control.Auto_Start,
                           R := "Station_Sys".Auto.Mode AND NOT "GluingControl".Control.Auto_Start,
                           PT := LT#10.7S);
END_REGION

REGION Network 4: Test
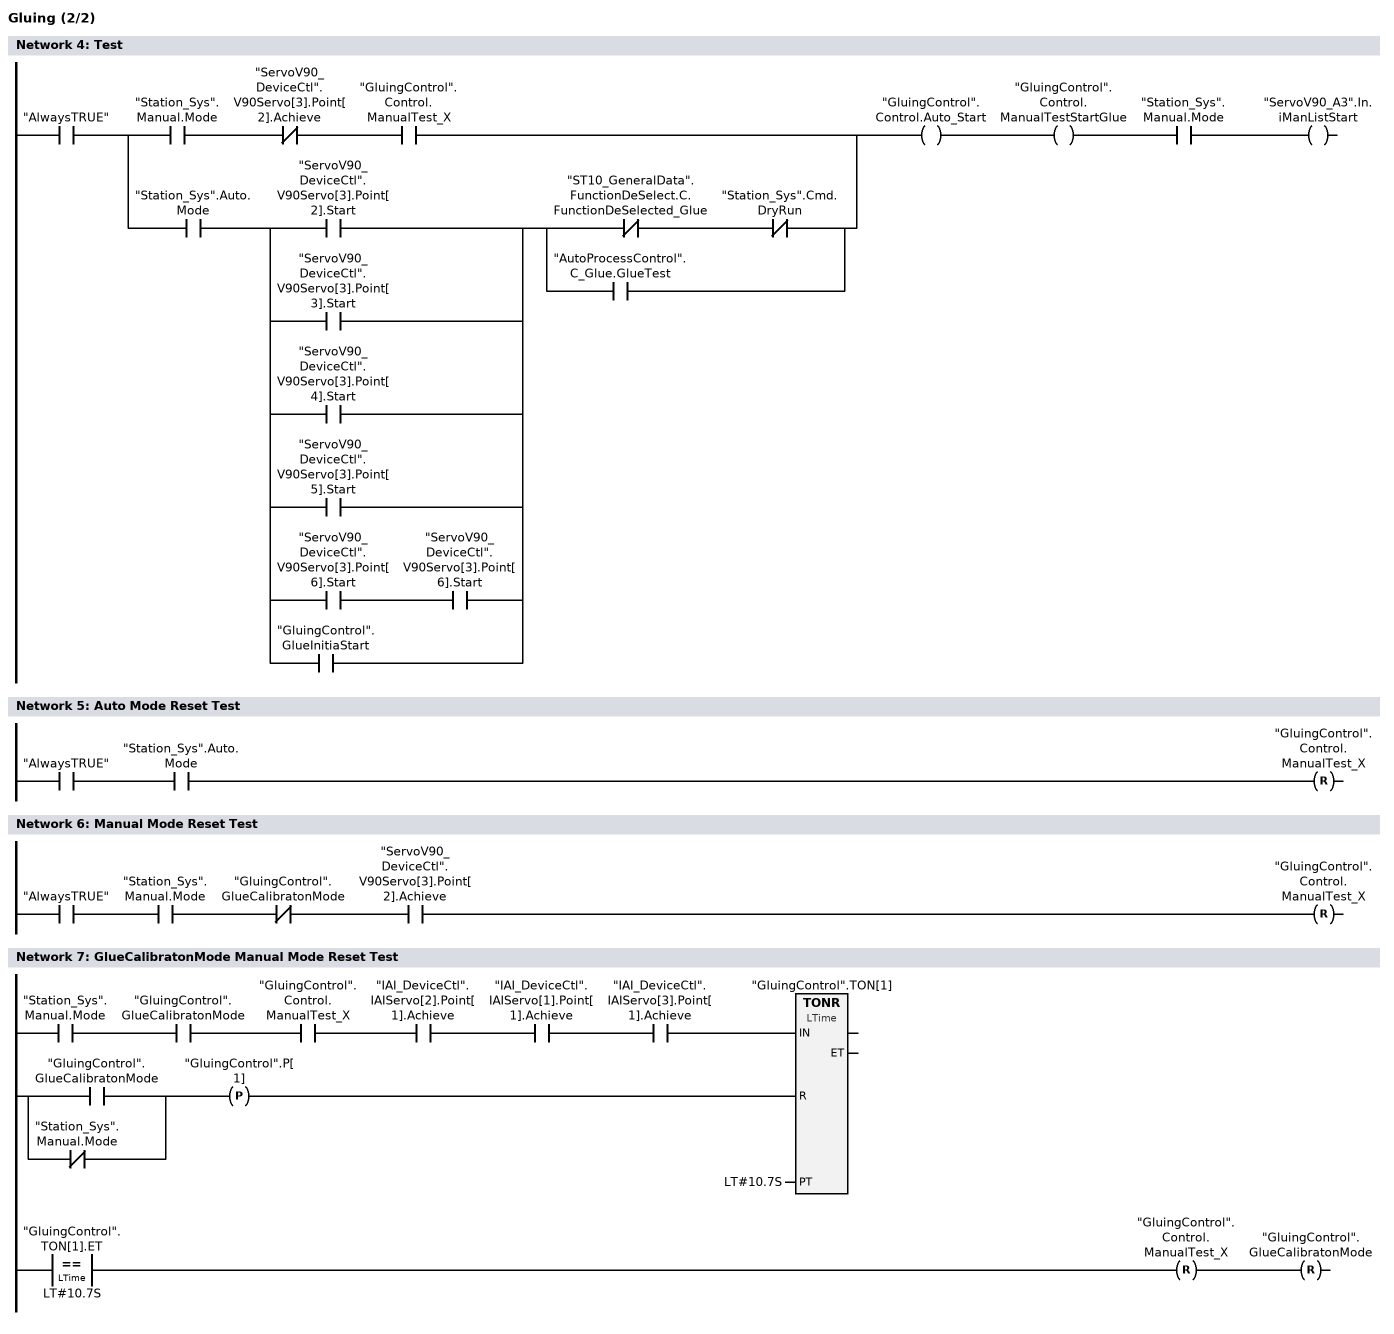
   RUNG wire#powerrail
      Contact( "AlwaysTRUE" )
      wire#w1
      Contact( "Station_Sys".Manual.Mode )
      I_Contact( "ServoV90_DeviceCtl".V90Servo[3].Point[2].Achieve )
      Contact( "GluingControl".Control.ManualTest_X )
      wire#w2
      Coil( "GluingControl".Control.Auto_Start )
      Coil( "GluingControl".Control.ManualTestStartGlue )
      Contact( "Station_Sys".Manual.Mode )
      Coil( "ServoV90_A3".In.iManListStart )
   END_RUNG
   RUNG wire#w1
      Contact( "Station_Sys".Auto.Mode )
      wire#w3
      Contact( "ServoV90_DeviceCtl".V90Servo[3].Point[2].Start )
      wire#w4
      I_Contact( "ST10_GeneralData".FunctionDeSelect.C.FunctionDeSelected_Glue )
      I_Contact( "Station_Sys".Cmd.DryRun )
   END_RUNG wire#w2
   RUNG wire#w3
      Contact( "ServoV90_DeviceCtl".V90Servo[3].Point[3].Start )
   END_RUNG wire#w4
   RUNG wire#w3
      Contact( "ServoV90_DeviceCtl".V90Servo[3].Point[4].Start )
   END_RUNG wire#w4
   RUNG wire#w3
      Contact( "ServoV90_DeviceCtl".V90Servo[3].Point[5].Start )
   END_RUNG wire#w4
   RUNG wire#w3
      Contact( "ServoV90_DeviceCtl".V90Servo[3].Point[6].Start )
      Contact( "ServoV90_DeviceCtl".V90Servo[3].Point[6].Start )
   END_RUNG wire#w4
   RUNG wire#w3
      Contact( "GluingControl".GlueInitiaStart )
   END_RUNG wire#w4
   RUNG wire#w4
      Contact( "AutoProcessControl".C_Glue.GlueTest )
   END_RUNG wire#w2
   // the same network as SCL:
   "GluingControl".Control.Auto_Start := "AlwaysTRUE" AND (("Station_Sys".Manual.Mode AND NOT "ServoV90_DeviceCtl".V90Servo[3].Point[2].Achieve AND "GluingControl".Control.ManualTest_X) OR ("Station_Sys".Auto.Mode AND ("ServoV90_DeviceCtl".V90Servo[3].Point[2].Start OR "ServoV90_DeviceCtl".V90Servo[3].Point[3].Start OR "ServoV90_DeviceCtl".V90Servo[3].Point[4].Start OR "ServoV90_DeviceCtl".V90Servo[3].Point[5].Start OR ("ServoV90_DeviceCtl".V90Servo[3].Point[6].Start AND "ServoV90_DeviceCtl".V90Servo[3].Point[6].Start) OR "GluingControl".GlueInitiaStart) AND ((NOT "ST10_GeneralData".FunctionDeSelect.C.FunctionDeSelected_Glue AND NOT "Station_Sys".Cmd.DryRun) OR "AutoProcessControl".C_Glue.GlueTest)));
   "GluingControl".Control.ManualTestStartGlue := "GluingControl".Control.Auto_Start;
   "ServoV90_A3".In.iManListStart := "GluingControl".Control.Auto_Start AND "Station_Sys".Manual.Mode;
END_REGION

REGION Network 5: Auto Mode Reset Test
   RUNG wire#powerrail
      Contact( "AlwaysTRUE" )
      Contact( "Station_Sys".Auto.Mode )
      R_Coil( "GluingControl".Control.ManualTest_X )
   END_RUNG
   // the same network as SCL:
   IF "AlwaysTRUE" AND "Station_Sys".Auto.Mode THEN "GluingControl".Control.ManualTest_X := FALSE; END_IF;
END_REGION

REGION Network 6: Manual Mode Reset Test
   RUNG wire#powerrail
      Contact( "AlwaysTRUE" )
      Contact( "Station_Sys".Manual.Mode )
      I_Contact( "GluingControl".GlueCalibratonMode )
      Contact( "ServoV90_DeviceCtl".V90Servo[3].Point[2].Achieve )
      R_Coil( "GluingControl".Control.ManualTest_X )
   END_RUNG
   // the same network as SCL:
   IF "AlwaysTRUE" AND "Station_Sys".Manual.Mode AND NOT "GluingControl".GlueCalibratonMode AND "ServoV90_DeviceCtl".V90Servo[3].Point[2].Achieve THEN
       "GluingControl".Control.ManualTest_X := FALSE;
   END_IF;
END_REGION

